   1:  PR[91,1] = PR[90,1] + -30.117;
   1:  PR[91,2] = PR[90,2] + 6.840;
   1:  PR[91,3] = PR[90,3] + 34.185;
   1:L PR[91] R[100]mm/sec CNT100;
   1:  PR[91,1] = PR[90,1] + -30.437;
   1:  PR[91,2] = PR[90,2] + 5.969;
   1:  PR[91,3] = PR[90,3] + 34.192;
   1:L PR[91] R[100]mm/sec CNT100;
   1:  PR[91,1] = PR[90,1] + -30.709;
   1:  PR[91,2] = PR[90,2] + 5.090;
   1:  PR[91,3] = PR[90,3] + 34.200;
   1:L PR[91] R[100]mm/sec CNT100;
   1:  PR[91,1] = PR[90,1] + -30.933;
   1:  PR[91,2] = PR[90,2] + 4.203;
   1:  PR[91,3] = PR[90,3] + 34.207;
   1:L PR[91] R[100]mm/sec CNT100;
   1:  PR[91,1] = PR[90,1] + -31.107;
   1:  PR[91,2] = PR[90,2] + 3.301;
   1:  PR[91,3] = PR[90,3] + 34.214;
   1:L PR[91] R[100]mm/sec CNT100;
   1:  PR[91,1] = PR[90,1] + -31.232;
   1:  PR[91,2] = PR[90,2] + 2.376;
   1:  PR[91,3] = PR[90,3] + 34.221;
   1:L PR[91] R[100]mm/sec CNT100;
   1:  PR[91,1] = PR[90,1] + -31.307;
   1:  PR[91,2] = PR[90,2] + 1.420;
   1:  PR[91,3] = PR[90,3] + 34.229;
   1:L PR[91] R[100]mm/sec CNT100;
   1:  PR[91,1] = PR[90,1] + -31.333;
   1:  PR[91,2] = PR[90,2] + 0.428;
   1:  PR[91,3] = PR[90,3] + 34.236;
   1:L PR[91] R[100]mm/sec CNT100;
   1:  PR[91,1] = PR[90,1] + -31.307;
   1:  PR[91,2] = PR[90,2] + -0.565;
   1:  PR[91,3] = PR[90,3] + 34.244;
   1:L PR[91] R[100]mm/sec CNT100;
   1:  PR[91,1] = PR[90,1] + -31.232;
   1:  PR[91,2] = PR[90,2] + -1.521;
   1:  PR[91,3] = PR[90,3] + 34.252;
   1:L PR[91] R[100]mm/sec CNT100;
   1:  PR[91,1] = PR[90,1] + -31.107;
   1:  PR[91,2] = PR[90,2] + -2.446;
   1:  PR[91,3] = PR[90,3] + 34.259;
   1:L PR[91] R[100]mm/sec CNT100;
   1:  PR[91,1] = PR[90,1] + -30.933;
   1:  PR[91,2] = PR[90,2] + -3.348;
   1:  PR[91,3] = PR[90,3] + 34.267;
   1:L PR[91] R[100]mm/sec CNT100;
   1:  PR[91,1] = PR[90,1] + -30.709;
   1:  PR[91,2] = PR[90,2] + -4.235;
   1:  PR[91,3] = PR[90,3] + 34.274;
   1:L PR[91] R[100]mm/sec CNT100;
   1:  PR[91,1] = PR[90,1] + -30.437;
   1:  PR[91,2] = PR[90,2] + -5.114;
   1:  PR[91,3] = PR[90,3] + 34.281;
   1:L PR[91] R[100]mm/sec CNT100;
   1:  PR[91,1] = PR[90,1] + -30.117;
   1:  PR[91,2] = PR[90,2] + -5.985;
   1:  PR[91,3] = PR[90,3] + 34.288;
   1:L PR[91] R[100]mm/sec CNT100;
   1:  PR[91,1] = PR[90,1] + -29.750;
   1:  PR[91,2] = PR[90,2] + -6.850;
   1:  PR[91,3] = PR[90,3] + 34.296;
   1:L PR[91] R[100]mm/sec CNT100;
   1:  PR[91,1] = PR[90,1] + -29.338;
   1:  PR[91,2] = PR[90,2] + -7.703;
   1:  PR[91,3] = PR[90,3] + 34.303;
   1:L PR[91] R[100]mm/sec CNT100;
   1:  PR[91,1] = PR[90,1] + -28.881;
   1:  PR[91,2] = PR[90,2] + -8.539;
   1:  PR[91,3] = PR[90,3] + 34.311;
   1:L PR[91] R[100]mm/sec CNT100;
   1:  PR[91,1] = PR[90,1] + -28.381;
   1:  PR[91,2] = PR[90,2] + -9.354;
   1:  PR[91,3] = PR[90,3] + 34.318;
   1:L PR[91] R[100]mm/sec CNT100;
   1:  PR[91,1] = PR[90,1] + -27.841;
   1:  PR[91,2] = PR[90,2] + -10.142;
   1:  PR[91,3] = PR[90,3] + 34.326;
   1:L PR[91] R[100]mm/sec CNT100;
   1:  PR[91,1] = PR[90,1] + -27.254;
   1:  PR[91,2] = PR[90,2] + -10.910;
   1:  PR[91,3] = PR[90,3] + 34.333;
   1:L PR[91] R[100]mm/sec CNT100;
   1:  PR[91,1] = PR[90,1] + -26.623;
   1:  PR[91,2] = PR[90,2] + -11.651;
   1:  PR[91,3] = PR[90,3] + 34.341;
   1:L PR[91] R[100]mm/sec CNT100;
   1:  PR[91,1] = PR[90,1] + -25.951;
   1:  PR[91,2] = PR[90,2] + -12.362;
   1:  PR[91,3] = PR[90,3] + 34.349;
   1:L PR[91] R[100]mm/sec CNT100;
   1:  PR[91,1] = PR[90,1] + -25.240;
   1:  PR[91,2] = PR[90,2] + -13.041;
   1:  PR[91,3] = PR[90,3] + 34.356;
   1:L PR[91] R[100]mm/sec CNT100;
   1:  PR[91,1] = PR[90,1] + -24.491;
   1:  PR[91,2] = PR[90,2] + -13.687;
   1:  PR[91,3] = PR[90,3] + 34.364;
   1:L PR[91] R[100]mm/sec CNT100;
   1:  PR[91,1] = PR[90,1] + -23.938;
   1:  PR[91,2] = PR[90,2] + -14.118;
   1:  PR[91,3] = PR[90,3] + 34.372;
   1:L PR[91] R[100]mm/sec CNT100;
   1:  PR[91,1] = PR[90,1] + -23.708;
   1:  PR[91,2] = PR[90,2] + -14.295;
   1:  PR[91,3] = PR[90,3] + 34.377;
   1:L PR[91] R[100]mm/sec CNT100;
   1:  PR[91,1] = PR[90,1] + -22.887;
   1:  PR[91,2] = PR[90,2] + -14.869;
   1:  PR[91,3] = PR[90,3] + 34.380;
   1:L PR[91] R[100]mm/sec CNT100;
   1:  PR[91,1] = PR[90,1] + -22.035;
   1:  PR[91,2] = PR[90,2] + -15.404;
   1:  PR[91,3] = PR[90,3] + 34.388;
   1:L PR[91] R[100]mm/sec CNT100;
   1:  PR[91,1] = PR[90,1] + -21.152;
   1:  PR[91,2] = PR[90,2] + -15.899;
   1:  PR[91,3] = PR[90,3] + 34.396;
   1:L PR[91] R[100]mm/sec CNT100;
   1:  PR[91,1] = PR[90,1] + -20.241;
   1:  PR[91,2] = PR[90,2] + -16.352;
   1:  PR[91,3] = PR[90,3] + 34.404;
   1:L PR[91] R[100]mm/sec CNT100;
   1:  PR[91,1] = PR[90,1] + -19.305;
   1:  PR[91,2] = PR[90,2] + -16.760;
   1:  PR[91,3] = PR[90,3] + 34.412;
   1:L PR[91] R[100]mm/sec CNT100;
   1:  PR[91,1] = PR[90,1] + -18.345;
   1:  PR[91,2] = PR[90,2] + -17.123;
   1:  PR[91,3] = PR[90,3] + 34.420;
   1:L PR[91] R[100]mm/sec CNT100;
   1:  PR[91,1] = PR[90,1] + -17.364;
   1:  PR[91,2] = PR[90,2] + -17.438;
   1:  PR[91,3] = PR[90,3] + 34.428;
   1:L PR[91] R[100]mm/sec CNT100;
   1:  PR[91,1] = PR[90,1] + -16.364;
   1:  PR[91,2] = PR[90,2] + -17.705;
   1:  PR[91,3] = PR[90,3] + 34.436;
   1:L PR[91] R[100]mm/sec CNT100;
   1:  PR[91,1] = PR[90,1] + -15.349;
   1:  PR[91,2] = PR[90,2] + -17.922;
   1:  PR[91,3] = PR[90,3] + 34.444;
   1:L PR[91] R[100]mm/sec CNT100;
   1:  PR[91,1] = PR[90,1] + -14.308;
   1:  PR[91,2] = PR[90,2] + -18.090;
   1:  PR[91,3] = PR[90,3] + 34.452;
   1:L PR[91] R[100]mm/sec CNT100;
   1:  PR[91,1] = PR[90,1] + -13.316;
   1:  PR[91,2] = PR[90,2] + -18.202;
   1:  PR[91,3] = PR[90,3] + 34.461;
   1:L PR[91] R[100]mm/sec CNT100;
   1:  PR[91,1] = PR[90,1] + -12.315;
   1:  PR[91,2] = PR[90,2] + -18.266;
   1:  PR[91,3] = PR[90,3] + 34.468;
   1:L PR[91] R[100]mm/sec CNT100;
   1:  PR[91,1] = PR[90,1] + -11.313;
   1:  PR[91,2] = PR[90,2] + -18.282;
   1:  PR[91,3] = PR[90,3] + 34.476;
   1:L PR[91] R[100]mm/sec CNT100;
   1:  PR[91,1] = PR[90,1] + -10.312;
   1:  PR[91,2] = PR[90,2] + -18.250;
   1:  PR[91,3] = PR[90,3] + 34.484;
   1:L PR[91] R[100]mm/sec CNT100;
   1:  PR[91,1] = PR[90,1] + -9.313;
   1:  PR[91,2] = PR[90,2] + -18.169;
   1:  PR[91,3] = PR[90,3] + 34.492;
   1:L PR[91] R[100]mm/sec CNT100;
   1:  PR[91,1] = PR[90,1] + -8.321;
   1:  PR[91,2] = PR[90,2] + -18.039;
   1:  PR[91,3] = PR[90,3] + 34.500;
   1:L PR[91] R[100]mm/sec CNT100;
   1:  PR[91,1] = PR[90,1] + -7.337;
   1:  PR[91,2] = PR[90,2] + -17.862;
   1:  PR[91,3] = PR[90,3] + 34.508;
   1:L PR[91] R[100]mm/sec CNT100;
   1:  PR[91,1] = PR[90,1] + -6.364;
   1:  PR[91,2] = PR[90,2] + -17.636;
   1:  PR[91,3] = PR[90,3] + 34.516;
   1:L PR[91] R[100]mm/sec CNT100;
   1:  PR[91,1] = PR[90,1] + -5.403;
   1:  PR[91,2] = PR[90,2] + -17.363;
   1:  PR[91,3] = PR[90,3] + 34.524;
   1:L PR[91] R[100]mm/sec CNT100;
   1:  PR[91,1] = PR[90,1] + -4.840;
   1:  PR[91,2] = PR[90,2] + -17.177;
   1:  PR[91,3] = PR[90,3] + 34.532;
   1:L PR[91] R[100]mm/sec CNT100;
   1:  PR[91,1] = PR[90,1] + -3.848;
   1:  PR[91,2] = PR[90,2] + -16.806;
   1:  PR[91,3] = PR[90,3] + 34.536;
   1:L PR[91] R[100]mm/sec CNT100;
   1:  PR[91,1] = PR[90,1] + -2.883;
   1:  PR[91,2] = PR[90,2] + -16.387;
   1:  PR[91,3] = PR[90,3] + 34.545;
   1:L PR[91] R[100]mm/sec CNT100;
   1:  PR[91,1] = PR[90,1] + -1.942;
   1:  PR[91,2] = PR[90,2] + -15.918;
   1:  PR[91,3] = PR[90,3] + 34.553;
   1:L PR[91] R[100]mm/sec CNT100;
   1:  PR[91,1] = PR[90,1] + -1.554;
   1:  PR[91,2] = PR[90,2] + -15.705;
   1:  PR[91,3] = PR[90,3] + 34.561;
   1:L PR[91] R[100]mm/sec CNT100;
   1:  PR[91,1] = PR[90,1] + -1.132;
   1:  PR[91,2] = PR[90,2] + -15.511;
   1:  PR[91,3] = PR[90,3] + 34.565;
   1:L PR[91] R[100]mm/sec CNT100;
   1:  PR[91,1] = PR[90,1] + -0.658;
   1:  PR[91,2] = PR[90,2] + -15.382;
   1:  PR[91,3] = PR[90,3] + 34.568;
   1:L PR[91] R[100]mm/sec CNT100;
   1:  PR[91,1] = PR[90,1] + -0.170;
   1:  PR[91,2] = PR[90,2] + -15.334;
   1:  PR[91,3] = PR[90,3] + 34.572;
   1:L PR[91] R[100]mm/sec CNT100;
   1:  PR[91,1] = PR[90,1] + 0.322;
   1:  PR[91,2] = PR[90,2] + -15.366;
   1:  PR[91,3] = PR[90,3] + 34.576;
   1:L PR[91] R[100]mm/sec CNT100;
   1:  PR[91] = PR[90];
   1:  PR[91,1] = PR[90,1] + 0.880;
   1:  PR[91,2] = PR[90,2] + -15.981;
   1:  PR[91,3] = PR[90,3] + 35.910;
   1:L PR[91] R[100]mm/sec CNT100;
   1:  PR[91,1] = PR[90,1] + 1.236;
   1:  PR[91,2] = PR[90,2] + -16.136;
   1:  PR[91,3] = PR[90,3] + 34.584;
   1:L PR[91] R[100]mm/sec CNT100;
   1:  PR[91,1] = PR[90,1] + 1.910;
   1:  PR[91,2] = PR[90,2] + -16.474;
   1:  PR[91,3] = PR[90,3] + 34.587;
   1:L PR[91] R[100]mm/sec CNT100;
   1:  PR[91,1] = PR[90,1] + 2.739;
   1:  PR[91,2] = PR[90,2] + -16.844;
   1:  PR[91,3] = PR[90,3] + 34.593;
   1:L PR[91] R[100]mm/sec CNT100;
   1:  PR[91,1] = PR[90,1] + 3.804;
   1:  PR[91,2] = PR[90,2] + -17.258;
   1:  PR[91,3] = PR[90,3] + 34.600;
   1:L PR[91] R[100]mm/sec CNT100;
   1:  PR[91,1] = PR[90,1] + 4.756;
   1:  PR[91,2] = PR[90,2] + -17.571;
   1:  PR[91,3] = PR[90,3] + 34.609;
   1:L PR[91] R[100]mm/sec CNT100;
   1:  PR[91,1] = PR[90,1] + 5.722;
   1:  PR[91,2] = PR[90,2] + -17.837;
   1:  PR[91,3] = PR[90,3] + 34.617;
   1:L PR[91] R[100]mm/sec CNT100;
   1:  PR[91,1] = PR[90,1] + 6.804;
   1:  PR[91,2] = PR[90,2] + -18.077;
   1:  PR[91,3] = PR[90,3] + 34.625;
   1:L PR[91] R[100]mm/sec CNT100;
   1:  PR[91,1] = PR[90,1] + 7.689;
   1:  PR[91,2] = PR[90,2] + -18.229;
   1:  PR[91,3] = PR[90,3] + 34.634;
   1:L PR[91] R[100]mm/sec CNT100;
   1:  PR[91,1] = PR[90,1] + 8.683;
   1:  PR[91,2] = PR[90,2] + -18.352;
   1:  PR[91,3] = PR[90,3] + 34.641;
   1:L PR[91] R[100]mm/sec CNT100;
   1:  PR[91,1] = PR[90,1] + 9.992;
   1:  PR[91,2] = PR[90,2] + -18.438;
   1:  PR[91,3] = PR[90,3] + 34.649;
   1:L PR[91] R[100]mm/sec CNT100;
   1:  PR[91,1] = PR[90,1] + 10.692;
   1:  PR[91,2] = PR[90,2] + -18.454;
   1:  PR[91,3] = PR[90,3] + 34.660;
   1:L PR[91] R[100]mm/sec CNT100;
   1:  PR[91,1] = PR[90,1] + 11.698;
   1:  PR[91,2] = PR[90,2] + -18.431;
   1:  PR[91,3] = PR[90,3] + 34.665;
   1:L PR[91] R[100]mm/sec CNT100;
   1:  PR[91,1] = PR[90,1] + 12.702;
   1:  PR[91,2] = PR[90,2] + -18.360;
   1:  PR[91,3] = PR[90,3] + 34.673;
   1:L PR[91] R[100]mm/sec CNT100;
   1:  PR[91,1] = PR[90,1] + 13.700;
   1:  PR[91,2] = PR[90,2] + -18.241;
   1:  PR[91,3] = PR[90,3] + 34.681;
   1:L PR[91] R[100]mm/sec CNT100;
   1:  PR[91,1] = PR[90,1] + 14.691;
   1:  PR[91,2] = PR[90,2] + -18.073;
   1:  PR[91,3] = PR[90,3] + 34.689;
   1:L PR[91] R[100]mm/sec CNT100;
   1:  PR[91,1] = PR[90,1] + 15.673;
   1:  PR[91,2] = PR[90,2] + -17.858;
   1:  PR[91,3] = PR[90,3] + 34.697;
   1:L PR[91] R[100]mm/sec CNT100;
   1:  PR[91,1] = PR[90,1] + 16.643;
   1:  PR[91,2] = PR[90,2] + -17.595;
   1:  PR[91,3] = PR[90,3] + 34.705;
   1:L PR[91] R[100]mm/sec CNT100;
   1:  PR[91,1] = PR[90,1] + 17.597;
   1:  PR[91,2] = PR[90,2] + -17.287;
   1:  PR[91,3] = PR[90,3] + 34.713;
   1:L PR[91] R[100]mm/sec CNT100;
   1:  PR[91,1] = PR[90,1] + 18.535;
   1:  PR[91,2] = PR[90,2] + -16.932;
   1:  PR[91,3] = PR[90,3] + 34.721;
   1:L PR[91] R[100]mm/sec CNT100;
   1:  PR[91,1] = PR[90,1] + 19.454;
   1:  PR[91,2] = PR[90,2] + -16.534;
   1:  PR[91,3] = PR[90,3] + 34.729;
   1:L PR[91] R[100]mm/sec CNT100;
   1:  PR[91,1] = PR[90,1] + 20.350;
   1:  PR[91,2] = PR[90,2] + -16.093;
   1:  PR[91,3] = PR[90,3] + 34.737;
   1:L PR[91] R[100]mm/sec CNT100;
   1:  PR[91,1] = PR[90,1] + 21.242;
   1:  PR[91,2] = PR[90,2] + -15.600;
   1:  PR[91,3] = PR[90,3] + 34.745;
   1:L PR[91] R[100]mm/sec CNT100;
   1:  PR[91,1] = PR[90,1] + 22.108;
   1:  PR[91,2] = PR[90,2] + -15.063;
   1:  PR[91,3] = PR[90,3] + 34.753;
   1:L PR[91] R[100]mm/sec CNT100;
   1:  PR[91,1] = PR[90,1] + 22.940;
   1:  PR[91,2] = PR[90,2] + -14.487;
   1:  PR[91,3] = PR[90,3] + 34.761;
   1:L PR[91] R[100]mm/sec CNT100;
   1:  PR[91,1] = PR[90,1] + 23.738;
   1:  PR[91,2] = PR[90,2] + -13.872;
   1:  PR[91,3] = PR[90,3] + 34.769;
   1:L PR[91] R[100]mm/sec CNT100;
   1:  PR[91,1] = PR[90,1] + 24.292;
   1:  PR[91,2] = PR[90,2] + -13.400;
   1:  PR[91,3] = PR[90,3] + 34.777;
   1:L PR[91] R[100]mm/sec CNT100;
   1:  PR[91,1] = PR[90,1] + 25.224;
   1:  PR[91,2] = PR[90,2] + -12.533;
   1:  PR[91,3] = PR[90,3] + 34.783;
   1:L PR[91] R[100]mm/sec CNT100;
   1:  PR[91,1] = PR[90,1] + 25.905;
   1:  PR[91,2] = PR[90,2] + -11.814;
   1:  PR[91,3] = PR[90,3] + 34.793;
   1:L PR[91] R[100]mm/sec CNT100;
   1:  PR[91,1] = PR[90,1] + 26.547;
   1:  PR[91,2] = PR[90,2] + -11.061;
   1:  PR[91,3] = PR[90,3] + 34.801;
   1:L PR[91] R[100]mm/sec CNT100;
   1:  PR[91,1] = PR[90,1] + 27.147;
   1:  PR[91,2] = PR[90,2] + -10.279;
   1:  PR[91,3] = PR[90,3] + 34.809;
   1:L PR[91] R[100]mm/sec CNT100;
   1:  PR[91,1] = PR[90,1] + 27.703;
   1:  PR[91,2] = PR[90,2] + -9.470;
   1:  PR[91,3] = PR[90,3] + 34.817;
   1:L PR[91] R[100]mm/sec CNT100;
   1:  PR[91,1] = PR[90,1] + 28.215;
   1:  PR[91,2] = PR[90,2] + -8.638;
   1:  PR[91,3] = PR[90,3] + 34.825;
   1:L PR[91] R[100]mm/sec CNT100;
   1:  PR[91,1] = PR[90,1] + 28.681;
   1:  PR[91,2] = PR[90,2] + -7.788;
   1:  PR[91,3] = PR[90,3] + 34.833;
   1:L PR[91] R[100]mm/sec CNT100;
   1:  PR[91,1] = PR[90,1] + 29.101;
   1:  PR[91,2] = PR[90,2] + -6.925;
   1:  PR[91,3] = PR[90,3] + 34.840;
   1:L PR[91] R[100]mm/sec CNT100;
   1:  PR[91,1] = PR[90,1] + 29.472;
   1:  PR[91,2] = PR[90,2] + -6.053;
   1:  PR[91,3] = PR[90,3] + 34.848;
   1:L PR[91] R[100]mm/sec CNT100;
   1:  PR[91,1] = PR[90,1] + 29.795;
   1:  PR[91,2] = PR[90,2] + -5.175;
   1:  PR[91,3] = PR[90,3] + 34.855;
   1:L PR[91] R[100]mm/sec CNT100;
   1:  PR[91,1] = PR[90,1] + 30.069;
   1:  PR[91,2] = PR[90,2] + -4.288;
   1:  PR[91,3] = PR[90,3] + 34.863;
   1:L PR[91] R[100]mm/sec CNT100;
   1:  PR[91,1] = PR[90,1] + 30.293;
   1:  PR[91,2] = PR[90,2] + -3.390;
   1:  PR[91,3] = PR[90,3] + 34.870;
   1:L PR[91] R[100]mm/sec CNT100;
   1:  PR[91,1] = PR[90,1] + 30.468;
   1:  PR[91,2] = PR[90,2] + -2.475;
   1:  PR[91,3] = PR[90,3] + 34.878;
   1:L PR[91] R[100]mm/sec CNT100;
   1:  PR[91,1] = PR[90,1] + 30.593;
   1:  PR[91,2] = PR[90,2] + -1.537;
   1:  PR[91,3] = PR[90,3] + 34.885;
   1:L PR[91] R[100]mm/sec CNT100;
   1:  PR[91,1] = PR[90,1] + 30.669;
   1:  PR[91,2] = PR[90,2] + -0.572;
   1:  PR[91,3] = PR[90,3] + 34.893;
   1:L PR[91] R[100]mm/sec CNT100;
   1:  PR[91,1] = PR[90,1] + 30.692;
   1:  PR[91,2] = PR[90,2] + 0.428;
   1:  PR[91,3] = PR[90,3] + 34.900;
   1:L PR[91] R[100]mm/sec CNT100;
   1:  PR[91,1] = PR[90,1] + 30.669;
   1:  PR[91,2] = PR[90,2] + 1.427;
   1:  PR[91,3] = PR[90,3] + 34.908;
   1:L PR[91] R[100]mm/sec CNT100;
   1:  PR[91,1] = PR[90,1] + 30.593;
   1:  PR[91,2] = PR[90,2] + 2.392;
   1:  PR[91,3] = PR[90,3] + 34.916;
   1:L PR[91] R[100]mm/sec CNT100;
   1:  PR[91,1] = PR[90,1] + 30.468;
   1:  PR[91,2] = PR[90,2] + 3.330;
   1:  PR[91,3] = PR[90,3] + 34.924;
   1:L PR[91] R[100]mm/sec CNT100;
   1:  PR[91,1] = PR[90,1] + 30.293;
   1:  PR[91,2] = PR[90,2] + 4.245;
   1:  PR[91,3] = PR[90,3] + 34.931;
   1:L PR[91] R[100]mm/sec CNT100;
   1:  PR[91,1] = PR[90,1] + 30.069;
   1:  PR[91,2] = PR[90,2] + 5.143;
   1:  PR[91,3] = PR[90,3] + 34.939;
   1:L PR[91] R[100]mm/sec CNT100;
   1:  PR[91,1] = PR[90,1] + 29.795;
   1:  PR[91,2] = PR[90,2] + 6.030;
   1:  PR[91,3] = PR[90,3] + 34.946;
   1:L PR[91] R[100]mm/sec CNT100;
   1:  PR[91,1] = PR[90,1] + 29.472;
   1:  PR[91,2] = PR[90,2] + 6.909;
   1:  PR[91,3] = PR[90,3] + 34.954;
   1:L PR[91] R[100]mm/sec CNT100;
   1:  PR[91,1] = PR[90,1] + 29.101;
   1:  PR[91,2] = PR[90,2] + 7.780;
   1:  PR[91,3] = PR[90,3] + 34.961;
   1:L PR[91] R[100]mm/sec CNT100;
   1:  PR[91,1] = PR[90,1] + 28.681;
   1:  PR[91,2] = PR[90,2] + 8.644;
   1:  PR[91,3] = PR[90,3] + 34.969;
   1:L PR[91] R[100]mm/sec CNT100;
   1:  PR[91,1] = PR[90,1] + 28.215;
   1:  PR[91,2] = PR[90,2] + 9.493;
   1:  PR[91,3] = PR[90,3] + 34.976;
   1:L PR[91] R[100]mm/sec CNT100;
   1:  PR[91,1] = PR[90,1] + 27.703;
   1:  PR[91,2] = PR[90,2] + 10.326;
   1:  PR[91,3] = PR[90,3] + 34.984;
   1:L PR[91] R[100]mm/sec CNT100;
   1:  PR[91,1] = PR[90,1] + 27.423;
   1:  PR[91,2] = PR[90,2] + 10.735;
   1:  PR[91,3] = PR[90,3] + 34.992;
   1:L PR[91] R[100]mm/sec CNT100;
   1:  PR[91,1] = PR[90,1] + 27.148;
   1:  PR[91,2] = PR[90,2] + 11.133;
   1:  PR[91,3] = PR[90,3] + 34.996;
   1:L PR[91] R[100]mm/sec CNT100;
   1:  PR[91,1] = PR[90,1] + 26.547;
   1:  PR[91,2] = PR[90,2] + 11.916;
   1:  PR[91,3] = PR[90,3] + 35.000;
   1:L PR[91] R[100]mm/sec CNT100;
   1:  PR[91,1] = PR[90,1] + 25.905;
   1:  PR[91,2] = PR[90,2] + 12.669;
   1:  PR[91,3] = PR[90,3] + 35.007;
   1:L PR[91] R[100]mm/sec CNT100;
   1:  PR[91,1] = PR[90,1] + 25.224;
   1:  PR[91,2] = PR[90,2] + 13.388;
   1:  PR[91,3] = PR[90,3] + 35.015;
   1:L PR[91] R[100]mm/sec CNT100;
   1:  PR[91,1] = PR[90,1] + 24.292;
   1:  PR[91,2] = PR[90,2] + 14.256;
   1:  PR[91,3] = PR[90,3] + 35.023;
   1:L PR[91] R[100]mm/sec CNT100;
   1:  PR[91,1] = PR[90,1] + 23.738;
   1:  PR[91,2] = PR[90,2] + 14.727;
   1:  PR[91,3] = PR[90,3] + 35.033;
   1:L PR[91] R[100]mm/sec CNT100;
   1:  PR[91,1] = PR[90,1] + 22.940;
   1:  PR[91,2] = PR[90,2] + 15.342;
   1:  PR[91,3] = PR[90,3] + 35.039;
   1:L PR[91] R[100]mm/sec CNT100;
   1:  PR[91,1] = PR[90,1] + 22.108;
   1:  PR[91,2] = PR[90,2] + 15.918;
   1:  PR[91,3] = PR[90,3] + 35.047;
   1:L PR[91] R[100]mm/sec CNT100;
   1:  PR[91,1] = PR[90,1] + 21.242;
   1:  PR[91,2] = PR[90,2] + 16.455;
   1:  PR[91,3] = PR[90,3] + 35.055;
   1:L PR[91] R[100]mm/sec CNT100;
   1:  PR[91,1] = PR[90,1] + 20.339;
   1:  PR[91,2] = PR[90,2] + 16.954;
   1:  PR[91,3] = PR[90,3] + 35.063;
   1:L PR[91] R[100]mm/sec CNT100;
   1:  PR[91,1] = PR[90,1] + 19.454;
   1:  PR[91,2] = PR[90,2] + 17.389;
   1:  PR[91,3] = PR[90,3] + 35.072;
   1:L PR[91] R[100]mm/sec CNT100;
   1:  PR[91,1] = PR[90,1] + 18.535;
   1:  PR[91,2] = PR[90,2] + 17.788;
   1:  PR[91,3] = PR[90,3] + 35.079;
   1:L PR[91] R[100]mm/sec CNT100;
   1:  PR[91,1] = PR[90,1] + 17.597;
   1:  PR[91,2] = PR[90,2] + 18.142;
   1:  PR[91,3] = PR[90,3] + 35.087;
   1:L PR[91] R[100]mm/sec CNT100;
   1:  PR[91,1] = PR[90,1] + 16.642;
   1:  PR[91,2] = PR[90,2] + 18.451;
   1:  PR[91,3] = PR[90,3] + 35.095;
   1:L PR[91] R[100]mm/sec CNT100;
   1:  PR[91,1] = PR[90,1] + 15.673;
   1:  PR[91,2] = PR[90,2] + 18.713;
   1:  PR[91,3] = PR[90,3] + 35.103;
   1:L PR[91] R[100]mm/sec CNT100;
   1:  PR[91,1] = PR[90,1] + 14.691;
   1:  PR[91,2] = PR[90,2] + 18.929;
   1:  PR[91,3] = PR[90,3] + 35.111;
   1:L PR[91] R[100]mm/sec CNT100;
   1:  PR[91,1] = PR[90,1] + 13.698;
   1:  PR[91,2] = PR[90,2] + 19.096;
   1:  PR[91,3] = PR[90,3] + 35.119;
   1:L PR[91] R[100]mm/sec CNT100;
   1:  PR[91,1] = PR[90,1] + 13.203;
   1:  PR[91,2] = PR[90,2] + 19.159;
   1:  PR[91,3] = PR[90,3] + 35.127;
   1:L PR[91] R[100]mm/sec CNT100;
   1:  PR[91,1] = PR[90,1] + 12.701;
   1:  PR[91,2] = PR[90,2] + 19.215;
   1:  PR[91,3] = PR[90,3] + 35.131;
   1:L PR[91] R[100]mm/sec CNT100;
   1:  PR[91,1] = PR[90,1] + 12.138;
   1:  PR[91,2] = PR[90,2] + 19.258;
   1:  PR[91,3] = PR[90,3] + 35.135;
   1:L PR[91] R[100]mm/sec CNT100;
   1:  PR[91,1] = PR[90,1] + 11.052;
   1:  PR[91,2] = PR[90,2] + 19.304;
   1:  PR[91,3] = PR[90,3] + 35.140;
   1:L PR[91] R[100]mm/sec CNT100;
   1:  PR[91,1] = PR[90,1] + 10.694;
   1:  PR[91,2] = PR[90,2] + 19.309;
   1:  PR[91,3] = PR[90,3] + 35.148;
   1:L PR[91] R[100]mm/sec CNT100;
   1:  PR[91,1] = PR[90,1] + 9.685;
   1:  PR[91,2] = PR[90,2] + 19.283;
   1:  PR[91,3] = PR[90,3] + 35.151;
   1:L PR[91] R[100]mm/sec CNT100;
   1:  PR[91,1] = PR[90,1] + 8.920;
   1:  PR[91,2] = PR[90,2] + 19.228;
   1:  PR[91,3] = PR[90,3] + 35.159;
   1:L PR[91] R[100]mm/sec CNT100;
   1:  PR[91,1] = PR[90,1] + 7.686;
   1:  PR[91,2] = PR[90,2] + 19.084;
   1:  PR[91,3] = PR[90,3] + 35.165;
   1:L PR[91] R[100]mm/sec CNT100;
   1:  PR[91,1] = PR[90,1] + 6.699;
   1:  PR[91,2] = PR[90,2] + 18.912;
   1:  PR[91,3] = PR[90,3] + 35.175;
   1:L PR[91] R[100]mm/sec CNT100;
   1:  PR[91,1] = PR[90,1] + 5.721;
   1:  PR[91,2] = PR[90,2] + 18.692;
   1:  PR[91,3] = PR[90,3] + 35.183;
   1:L PR[91] R[100]mm/sec CNT100;
   1:  PR[91,1] = PR[90,1] + 4.734;
   1:  PR[91,2] = PR[90,2] + 18.419;
   1:  PR[91,3] = PR[90,3] + 35.191;
   1:L PR[91] R[100]mm/sec CNT100;
   1:  PR[91,1] = PR[90,1] + 3.800;
   1:  PR[91,2] = PR[90,2] + 18.112;
   1:  PR[91,3] = PR[90,3] + 35.199;
   1:L PR[91] R[100]mm/sec CNT100;
   1:  PR[91,1] = PR[90,1] + 2.864;
   1:  PR[91,2] = PR[90,2] + 17.752;
   1:  PR[91,3] = PR[90,3] + 35.207;
   1:L PR[91] R[100]mm/sec CNT100;
   1:  PR[91,1] = PR[90,1] + 1.949;
   1:  PR[91,2] = PR[90,2] + 17.348;
   1:  PR[91,3] = PR[90,3] + 35.215;
   1:L PR[91] R[100]mm/sec CNT100;
   1:  PR[91,1] = PR[90,1] + 1.236;
   1:  PR[91,2] = PR[90,2] + 16.992;
   1:  PR[91,3] = PR[90,3] + 35.223;
   1:L PR[91] R[100]mm/sec CNT100;
   1:  PR[91,1] = PR[90,1] + 0.880;
   1:  PR[91,2] = PR[90,2] + 16.836;
   1:  PR[91,3] = PR[90,3] + 35.230;
   1:L PR[91] R[100]mm/sec CNT100;
   1:  PR[91,1] = PR[90,1] + 0.406;
   1:  PR[91,2] = PR[90,2] + 16.707;
   1:  PR[91,3] = PR[90,3] + 35.233;
   1:L PR[91] R[100]mm/sec CNT100;
   1:  PR[91,1] = PR[90,1] + -0.086;
   1:  PR[91,2] = PR[90,2] + 16.662;
   1:  PR[91,3] = PR[90,3] + 35.237;
   1:L PR[91] R[100]mm/sec CNT100;
   1:  PR[91,1] = PR[90,1] + -0.574;
   1:  PR[91,2] = PR[90,2] + 16.697;
   1:  PR[91,3] = PR[90,3] + 35.241;
   1:L PR[91] R[100]mm/sec CNT100;
   1:  PR[91,1] = PR[90,1] + -1.051;
   1:  PR[91,2] = PR[90,2] + 16.812;
   1:  PR[91,3] = PR[90,3] + 35.244;
   1:L PR[91] R[100]mm/sec CNT100;
   1:  PR[91,1] = PR[90,1] + -1.476;
   1:  PR[91,2] = PR[90,2] + 16.991;
   1:  PR[91,3] = PR[90,3] + 35.248;
   1:L PR[91] R[100]mm/sec CNT100;
   1:  PR[91,1] = PR[90,1] + -2.136;
   1:  PR[91,2] = PR[90,2] + 17.322;
   1:  PR[91,3] = PR[90,3] + 35.252;
   1:L PR[91] R[100]mm/sec CNT100;
   1:  PR[91,1] = PR[90,1] + -2.980;
   1:  PR[91,2] = PR[90,2] + 17.700;
   1:  PR[91,3] = PR[90,3] + 35.258;
   1:L PR[91] R[100]mm/sec CNT100;
   1:  PR[91,1] = PR[90,1] + -4.044;
   1:  PR[91,2] = PR[90,2] + 18.115;
   1:  PR[91,3] = PR[90,3] + 35.265;
   1:L PR[91] R[100]mm/sec CNT100;
   1:  PR[91,1] = PR[90,1] + -4.996;
   1:  PR[91,2] = PR[90,2] + 18.428;
   1:  PR[91,3] = PR[90,3] + 35.274;
   1:L PR[91] R[100]mm/sec CNT100;
   1:  PR[91,1] = PR[90,1] + -5.962;
   1:  PR[91,2] = PR[90,2] + 18.694;
   1:  PR[91,3] = PR[90,3] + 35.282;
   1:L PR[91] R[100]mm/sec CNT100;
   1:  PR[91,1] = PR[90,1] + -7.044;
   1:  PR[91,2] = PR[90,2] + 18.933;
   1:  PR[91,3] = PR[90,3] + 35.290;
   1:L PR[91] R[100]mm/sec CNT100;
   1:  PR[91,1] = PR[90,1] + -7.929;
   1:  PR[91,2] = PR[90,2] + 19.085;
   1:  PR[91,3] = PR[90,3] + 35.299;
   1:L PR[91] R[100]mm/sec CNT100;
   1:  PR[91,1] = PR[90,1] + -8.924;
   1:  PR[91,2] = PR[90,2] + 19.208;
   1:  PR[91,3] = PR[90,3] + 35.306;
   1:L PR[91] R[100]mm/sec CNT100;
   1:  PR[91,1] = PR[90,1] + -10.233;
   1:  PR[91,2] = PR[90,2] + 19.293;
   1:  PR[91,3] = PR[90,3] + 35.314;
   1:L PR[91] R[100]mm/sec CNT100;
   1:  PR[91,1] = PR[90,1] + -10.933;
   1:  PR[91,2] = PR[90,2] + 19.309;
   1:  PR[91,3] = PR[90,3] + 35.325;
   1:L PR[91] R[100]mm/sec CNT100;
   1:  PR[91,1] = PR[90,1] + -11.939;
   1:  PR[91,2] = PR[90,2] + 19.286;
   1:  PR[91,3] = PR[90,3] + 35.330;
   1:L PR[91] R[100]mm/sec CNT100;
   1:  PR[91,1] = PR[90,1] + -12.943;
   1:  PR[91,2] = PR[90,2] + 19.215;
   1:  PR[91,3] = PR[90,3] + 35.338;
   1:L PR[91] R[100]mm/sec CNT100;
   1:  PR[91,1] = PR[90,1] + -13.941;
   1:  PR[91,2] = PR[90,2] + 19.095;
   1:  PR[91,3] = PR[90,3] + 35.346;
   1:L PR[91] R[100]mm/sec CNT100;
   1:  PR[91,1] = PR[90,1] + -14.933;
   1:  PR[91,2] = PR[90,2] + 18.928;
   1:  PR[91,3] = PR[90,3] + 35.354;
   1:L PR[91] R[100]mm/sec CNT100;
   1:  PR[91,1] = PR[90,1] + -15.916;
   1:  PR[91,2] = PR[90,2] + 18.713;
   1:  PR[91,3] = PR[90,3] + 35.362;
   1:L PR[91] R[100]mm/sec CNT100;
   1:  PR[91,1] = PR[90,1] + -16.602;
   1:  PR[91,2] = PR[90,2] + 18.530;
   1:  PR[91,3] = PR[90,3] + 35.370;
   1:L PR[91] R[100]mm/sec CNT100;
   1:  PR[91,1] = PR[90,1] + -17.842;
   1:  PR[91,2] = PR[90,2] + 18.141;
   1:  PR[91,3] = PR[90,3] + 35.376;
   1:L PR[91] R[100]mm/sec CNT100;
   1:  PR[91,1] = PR[90,1] + -18.635;
   1:  PR[91,2] = PR[90,2] + 17.843;
   1:  PR[91,3] = PR[90,3] + 35.386;
   1:L PR[91] R[100]mm/sec CNT100;
   1:  PR[91,1] = PR[90,1] + -19.695;
   1:  PR[91,2] = PR[90,2] + 17.388;
   1:  PR[91,3] = PR[90,3] + 35.393;
   1:L PR[91] R[100]mm/sec CNT100;
   1:  PR[91,1] = PR[90,1] + -20.591;
   1:  PR[91,2] = PR[90,2] + 16.946;
   1:  PR[91,3] = PR[90,3] + 35.402;
   1:L PR[91] R[100]mm/sec CNT100;
   1:  PR[91,1] = PR[90,1] + -21.482;
   1:  PR[91,2] = PR[90,2] + 16.452;
   1:  PR[91,3] = PR[90,3] + 35.410;
   1:L PR[91] R[100]mm/sec CNT100;
   1:  PR[91,1] = PR[90,1] + -22.348;
   1:  PR[91,2] = PR[90,2] + 15.914;
   1:  PR[91,3] = PR[90,3] + 35.418;
   1:L PR[91] R[100]mm/sec CNT100;
   1:  PR[91,1] = PR[90,1] + -23.180;
   1:  PR[91,2] = PR[90,2] + 15.338;
   1:  PR[91,3] = PR[90,3] + 35.426;
   1:L PR[91] R[100]mm/sec CNT100;
   1:  PR[91,1] = PR[90,1] + -23.978;
   1:  PR[91,2] = PR[90,2] + 14.723;
   1:  PR[91,3] = PR[90,3] + 35.434;
   1:L PR[91] R[100]mm/sec CNT100;
   1:  PR[91,1] = PR[90,1] + -24.739;
   1:  PR[91,2] = PR[90,2] + 14.073;
   1:  PR[91,3] = PR[90,3] + 35.442;
   1:L PR[91] R[100]mm/sec CNT100;
   1:  PR[91,1] = PR[90,1] + -25.462;
   1:  PR[91,2] = PR[90,2] + 13.388;
   1:  PR[91,3] = PR[90,3] + 35.450;
   1:L PR[91] R[100]mm/sec CNT100;
   1:  PR[91,1] = PR[90,1] + -26.146;
   1:  PR[91,2] = PR[90,2] + 12.670;
   1:  PR[91,3] = PR[90,3] + 35.458;
   1:L PR[91] R[100]mm/sec CNT100;
   1:  PR[91,1] = PR[90,1] + -26.787;
   1:  PR[91,2] = PR[90,2] + 11.921;
   1:  PR[91,3] = PR[90,3] + 35.466;
   1:L PR[91] R[100]mm/sec CNT100;
   1:  PR[91,1] = PR[90,1] + -27.387;
   1:  PR[91,2] = PR[90,2] + 11.141;
   1:  PR[91,3] = PR[90,3] + 35.474;
   1:L PR[91] R[100]mm/sec CNT100;
   1:  PR[91,1] = PR[90,1] + -27.942;
   1:  PR[91,2] = PR[90,2] + 10.333;
   1:  PR[91,3] = PR[90,3] + 35.482;
   1:L PR[91] R[100]mm/sec CNT100;
   1:  PR[91,1] = PR[90,1] + -28.453;
   1:  PR[91,2] = PR[90,2] + 9.500;
   1:  PR[91,3] = PR[90,3] + 35.490;
   1:L PR[91] R[100]mm/sec CNT100;
   1:  PR[91,1] = PR[90,1] + -28.919;
   1:  PR[91,2] = PR[90,2] + 8.647;
   1:  PR[91,3] = PR[90,3] + 35.498;
   1:L PR[91] R[100]mm/sec CNT100;
   1:  PR[91,1] = PR[90,1] + -29.339;
   1:  PR[91,2] = PR[90,2] + 7.778;
   1:  PR[91,3] = PR[90,3] + 35.505;
   1:L PR[91] R[100]mm/sec CNT100;
   1:  PR[91,1] = PR[90,1] + -29.710;
   1:  PR[91,2] = PR[90,2] + 6.900;
   1:  PR[91,3] = PR[90,3] + 35.513;
   1:L PR[91] R[100]mm/sec CNT100;
   1:  PR[91,1] = PR[90,1] + -30.033;
   1:  PR[91,2] = PR[90,2] + 6.016;
   1:  PR[91,3] = PR[90,3] + 35.521;
   1:L PR[91] R[100]mm/sec CNT100;
   1:  PR[91,1] = PR[90,1] + -30.307;
   1:  PR[91,2] = PR[90,2] + 5.126;
   1:  PR[91,3] = PR[90,3] + 35.528;
   1:L PR[91] R[100]mm/sec CNT100;
   1:  PR[91,1] = PR[90,1] + -30.532;
   1:  PR[91,2] = PR[90,2] + 4.229;
   1:  PR[91,3] = PR[90,3] + 35.535;
   1:L PR[91] R[100]mm/sec CNT100;
   1:  PR[91,1] = PR[90,1] + -30.707;
   1:  PR[91,2] = PR[90,2] + 3.318;
   1:  PR[91,3] = PR[90,3] + 35.543;
   1:L PR[91] R[100]mm/sec CNT100;
   1:  PR[91,1] = PR[90,1] + -30.832;
   1:  PR[91,2] = PR[90,2] + 2.386;
   1:  PR[91,3] = PR[90,3] + 35.550;
   1:L PR[91] R[100]mm/sec CNT100;
   1:  PR[91,1] = PR[90,1] + -30.907;
   1:  PR[91,2] = PR[90,2] + 1.425;
   1:  PR[91,3] = PR[90,3] + 35.558;
   1:L PR[91] R[100]mm/sec CNT100;
   1:  PR[91,1] = PR[90,1] + -30.931;
   1:  PR[91,2] = PR[90,2] + 0.428;
   1:  PR[91,3] = PR[90,3] + 35.565;
   1:L PR[91] R[100]mm/sec CNT100;
   1:  PR[91,1] = PR[90,1] + -30.907;
   1:  PR[91,2] = PR[90,2] + -0.570;
   1:  PR[91,3] = PR[90,3] + 35.573;
   1:L PR[91] R[100]mm/sec CNT100;
   1:  PR[91,1] = PR[90,1] + -30.832;
   1:  PR[91,2] = PR[90,2] + -1.531;
   1:  PR[91,3] = PR[90,3] + 35.581;
   1:L PR[91] R[100]mm/sec CNT100;
   1:  PR[91,1] = PR[90,1] + -30.707;
   1:  PR[91,2] = PR[90,2] + -2.463;
   1:  PR[91,3] = PR[90,3] + 35.589;
   1:L PR[91] R[100]mm/sec CNT100;
   1:  PR[91,1] = PR[90,1] + -30.532;
   1:  PR[91,2] = PR[90,2] + -3.373;
   1:  PR[91,3] = PR[90,3] + 35.596;
   1:L PR[91] R[100]mm/sec CNT100;
   1:  PR[91,1] = PR[90,1] + -30.307;
   1:  PR[91,2] = PR[90,2] + -4.271;
   1:  PR[91,3] = PR[90,3] + 35.604;
   1:L PR[91] R[100]mm/sec CNT100;
   1:  PR[91,1] = PR[90,1] + -30.033;
   1:  PR[91,2] = PR[90,2] + -5.161;
   1:  PR[91,3] = PR[90,3] + 35.611;
   1:L PR[91] R[100]mm/sec CNT100;
   1:  PR[91,1] = PR[90,1] + -29.710;
   1:  PR[91,2] = PR[90,2] + -6.044;
   1:  PR[91,3] = PR[90,3] + 35.619;
   1:L PR[91] R[100]mm/sec CNT100;
   1:  PR[91,1] = PR[90,1] + -29.339;
   1:  PR[91,2] = PR[90,2] + -6.923;
   1:  PR[91,3] = PR[90,3] + 35.626;
   1:L PR[91] R[100]mm/sec CNT100;
   1:  PR[91,1] = PR[90,1] + -28.919;
   1:  PR[91,2] = PR[90,2] + -7.792;
   1:  PR[91,3] = PR[90,3] + 35.634;
   1:L PR[91] R[100]mm/sec CNT100;
   1:  PR[91,1] = PR[90,1] + -28.649;
   1:  PR[91,2] = PR[90,2] + -8.290;
   1:  PR[91,3] = PR[90,3] + 35.641;
   1:L PR[91] R[100]mm/sec CNT100;
   1:  PR[91,1] = PR[90,1] + -28.454;
   1:  PR[91,2] = PR[90,2] + -8.644;
   1:  PR[91,3] = PR[90,3] + 35.646;
   1:L PR[91] R[100]mm/sec CNT100;
   1:  PR[91,1] = PR[90,1] + -27.942;
   1:  PR[91,2] = PR[90,2] + -9.478;
   1:  PR[91,3] = PR[90,3] + 35.649;
   1:L PR[91] R[100]mm/sec CNT100;
   1:  PR[91,1] = PR[90,1] + -27.387;
   1:  PR[91,2] = PR[90,2] + -10.286;
   1:  PR[91,3] = PR[90,3] + 35.657;
   1:L PR[91] R[100]mm/sec CNT100;
   1:  PR[91,1] = PR[90,1] + -26.787;
   1:  PR[91,2] = PR[90,2] + -11.065;
   1:  PR[91,3] = PR[90,3] + 35.665;
   1:L PR[91] R[100]mm/sec CNT100;
   1:  PR[91,1] = PR[90,1] + -26.146;
   1:  PR[91,2] = PR[90,2] + -11.815;
   1:  PR[91,3] = PR[90,3] + 35.672;
   1:L PR[91] R[100]mm/sec CNT100;
   1:  PR[91,1] = PR[90,1] + -25.462;
   1:  PR[91,2] = PR[90,2] + -12.533;
   1:  PR[91,3] = PR[90,3] + 35.680;
   1:L PR[91] R[100]mm/sec CNT100;
   1:  PR[91,1] = PR[90,1] + -24.739;
   1:  PR[91,2] = PR[90,2] + -13.218;
   1:  PR[91,3] = PR[90,3] + 35.688;
   1:L PR[91] R[100]mm/sec CNT100;
   1:  PR[91,1] = PR[90,1] + -23.978;
   1:  PR[91,2] = PR[90,2] + -13.868;
   1:  PR[91,3] = PR[90,3] + 35.696;
   1:L PR[91] R[100]mm/sec CNT100;
   1:  PR[91,1] = PR[90,1] + -23.180;
   1:  PR[91,2] = PR[90,2] + -14.483;
   1:  PR[91,3] = PR[90,3] + 35.704;
   1:L PR[91] R[100]mm/sec CNT100;
   1:  PR[91,1] = PR[90,1] + -22.348;
   1:  PR[91,2] = PR[90,2] + -15.059;
   1:  PR[91,3] = PR[90,3] + 35.712;
   1:L PR[91] R[100]mm/sec CNT100;
   1:  PR[91,1] = PR[90,1] + -21.482;
   1:  PR[91,2] = PR[90,2] + -15.597;
   1:  PR[91,3] = PR[90,3] + 35.720;
   1:L PR[91] R[100]mm/sec CNT100;
   1:  PR[91,1] = PR[90,1] + -20.579;
   1:  PR[91,2] = PR[90,2] + -16.097;
   1:  PR[91,3] = PR[90,3] + 35.728;
   1:L PR[91] R[100]mm/sec CNT100;
   1:  PR[91,1] = PR[90,1] + -19.694;
   1:  PR[91,2] = PR[90,2] + -16.534;
   1:  PR[91,3] = PR[90,3] + 35.737;
   1:L PR[91] R[100]mm/sec CNT100;
   1:  PR[91,1] = PR[90,1] + -18.776;
   1:  PR[91,2] = PR[90,2] + -16.933;
   1:  PR[91,3] = PR[90,3] + 35.744;
   1:L PR[91] R[100]mm/sec CNT100;
   1:  PR[91,1] = PR[90,1] + -17.839;
   1:  PR[91,2] = PR[90,2] + -17.287;
   1:  PR[91,3] = PR[90,3] + 35.752;
   1:L PR[91] R[100]mm/sec CNT100;
   1:  PR[91,1] = PR[90,1] + -16.885;
   1:  PR[91,2] = PR[90,2] + -17.596;
   1:  PR[91,3] = PR[90,3] + 35.760;
   1:L PR[91] R[100]mm/sec CNT100;
   1:  PR[91,1] = PR[90,1] + -15.915;
   1:  PR[91,2] = PR[90,2] + -17.858;
   1:  PR[91,3] = PR[90,3] + 35.768;
   1:L PR[91] R[100]mm/sec CNT100;
   1:  PR[91,1] = PR[90,1] + -14.934;
   1:  PR[91,2] = PR[90,2] + -18.073;
   1:  PR[91,3] = PR[90,3] + 35.776;
   1:L PR[91] R[100]mm/sec CNT100;
   1:  PR[91,1] = PR[90,1] + -13.942;
   1:  PR[91,2] = PR[90,2] + -18.240;
   1:  PR[91,3] = PR[90,3] + 35.784;
   1:L PR[91] R[100]mm/sec CNT100;
   1:  PR[91,1] = PR[90,1] + -12.943;
   1:  PR[91,2] = PR[90,2] + -18.360;
   1:  PR[91,3] = PR[90,3] + 35.792;
   1:L PR[91] R[100]mm/sec CNT100;
   1:  PR[91,1] = PR[90,1] + -11.941;
   1:  PR[91,2] = PR[90,2] + -18.431;
   1:  PR[91,3] = PR[90,3] + 35.800;
   1:L PR[91] R[100]mm/sec CNT100;
   1:  PR[91,1] = PR[90,1] + -10.935;
   1:  PR[91,2] = PR[90,2] + -18.453;
   1:  PR[91,3] = PR[90,3] + 35.808;
   1:L PR[91] R[100]mm/sec CNT100;
   1:  PR[91,1] = PR[90,1] + -9.930;
   1:  PR[91,2] = PR[90,2] + -18.427;
   1:  PR[91,3] = PR[90,3] + 35.816;
   1:L PR[91] R[100]mm/sec CNT100;
   1:  PR[91,1] = PR[90,1] + -8.928;
   1:  PR[91,2] = PR[90,2] + -18.353;
   1:  PR[91,3] = PR[90,3] + 35.824;
   1:L PR[91] R[100]mm/sec CNT100;
   1:  PR[91,1] = PR[90,1] + -7.932;
   1:  PR[91,2] = PR[90,2] + -18.230;
   1:  PR[91,3] = PR[90,3] + 35.832;
   1:L PR[91] R[100]mm/sec CNT100;
   1:  PR[91,1] = PR[90,1] + -6.943;
   1:  PR[91,2] = PR[90,2] + -18.059;
   1:  PR[91,3] = PR[90,3] + 35.840;
   1:L PR[91] R[100]mm/sec CNT100;
   1:  PR[91,1] = PR[90,1] + -5.965;
   1:  PR[91,2] = PR[90,2] + -17.840;
   1:  PR[91,3] = PR[90,3] + 35.848;
   1:L PR[91] R[100]mm/sec CNT100;
   1:  PR[91,1] = PR[90,1] + -4.979;
   1:  PR[91,2] = PR[90,2] + -17.568;
   1:  PR[91,3] = PR[90,3] + 35.856;
   1:L PR[91] R[100]mm/sec CNT100;
   1:  PR[91,1] = PR[90,1] + -4.045;
   1:  PR[91,2] = PR[90,2] + -17.260;
   1:  PR[91,3] = PR[90,3] + 35.864;
   1:L PR[91] R[100]mm/sec CNT100;
   1:  PR[91,1] = PR[90,1] + -3.109;
   1:  PR[91,2] = PR[90,2] + -16.900;
   1:  PR[91,3] = PR[90,3] + 35.872;
   1:L PR[91] R[100]mm/sec CNT100;
   1:  PR[91,1] = PR[90,1] + -2.194;
   1:  PR[91,2] = PR[90,2] + -16.495;
   1:  PR[91,3] = PR[90,3] + 35.880;
   1:L PR[91] R[100]mm/sec CNT100;
   1:  PR[91,1] = PR[90,1] + -1.475;
   1:  PR[91,2] = PR[90,2] + -16.135;
   1:  PR[91,3] = PR[90,3] + 35.888;
   1:L PR[91] R[100]mm/sec CNT100;
   1:  PR[91,1] = PR[90,1] + -1.050;
   1:  PR[91,2] = PR[90,2] + -15.956;
   1:  PR[91,3] = PR[90,3] + 35.895;
   1:L PR[91] R[100]mm/sec CNT100;
   1:  PR[91,1] = PR[90,1] + -0.574;
   1:  PR[91,2] = PR[90,2] + -15.842;
   1:  PR[91,3] = PR[90,3] + 35.898;
   1:L PR[91] R[100]mm/sec CNT100;
   1:  PR[91,1] = PR[90,1] + -0.086;
   1:  PR[91,2] = PR[90,2] + -15.807;
   1:  PR[91,3] = PR[90,3] + 35.902;
   1:L PR[91] R[100]mm/sec CNT100;
   1:  PR[91,1] = PR[90,1] + 0.406;
   1:  PR[91,2] = PR[90,2] + -15.852;
   1:  PR[91,3] = PR[90,3] + 35.906;
   1:L PR[91] R[100]mm/sec CNT100;
   1:  PR[91] = PR[90];
   1:  PR[91,1] = PR[90,1] + 0.951;
   1:  PR[91,2] = PR[90,2] + -16.464;
   1:  PR[91,3] = PR[90,3] + 37.240;
   1:L PR[91] R[100]mm/sec CNT100;
   1:  PR[91,1] = PR[90,1] + 2.423;
   1:  PR[91,2] = PR[90,2] + -17.122;
   1:  PR[91,3] = PR[90,3] + 35.914;
   1:L PR[91] R[100]mm/sec CNT100;
   1:  PR[91,1] = PR[90,1] + 3.362;
   1:  PR[91,2] = PR[90,2] + -17.476;
   1:  PR[91,3] = PR[90,3] + 35.927;
   1:L PR[91] R[100]mm/sec CNT100;
   1:  PR[91,1] = PR[90,1] + 4.322;
   1:  PR[91,2] = PR[90,2] + -17.785;
   1:  PR[91,3] = PR[90,3] + 35.935;
   1:L PR[91] R[100]mm/sec CNT100;
   1:  PR[91,1] = PR[90,1] + 5.298;
   1:  PR[91,2] = PR[90,2] + -18.047;
   1:  PR[91,3] = PR[90,3] + 35.943;
   1:L PR[91] R[100]mm/sec CNT100;
   1:  PR[91,1] = PR[90,1] + 5.906;
   1:  PR[91,2] = PR[90,2] + -18.182;
   1:  PR[91,3] = PR[90,3] + 35.951;
   1:L PR[91] R[100]mm/sec CNT100;
   1:  PR[91,1] = PR[90,1] + 6.282;
   1:  PR[91,2] = PR[90,2] + -18.261;
   1:  PR[91,3] = PR[90,3] + 35.956;
   1:L PR[91] R[100]mm/sec CNT100;
   1:  PR[91,1] = PR[90,1] + 7.282;
   1:  PR[91,2] = PR[90,2] + -18.426;
   1:  PR[91,3] = PR[90,3] + 35.959;
   1:L PR[91] R[100]mm/sec CNT100;
   1:  PR[91,1] = PR[90,1] + 8.287;
   1:  PR[91,2] = PR[90,2] + -18.543;
   1:  PR[91,3] = PR[90,3] + 35.967;
   1:L PR[91] R[100]mm/sec CNT100;
   1:  PR[91,1] = PR[90,1] + 9.092;
   1:  PR[91,2] = PR[90,2] + -18.599;
   1:  PR[91,3] = PR[90,3] + 35.975;
   1:L PR[91] R[100]mm/sec CNT100;
   1:  PR[91,1] = PR[90,1] + 10.310;
   1:  PR[91,2] = PR[90,2] + -18.628;
   1:  PR[91,3] = PR[90,3] + 35.982;
   1:L PR[91] R[100]mm/sec CNT100;
   1:  PR[91,1] = PR[90,1] + 11.320;
   1:  PR[91,2] = PR[90,2] + -18.598;
   1:  PR[91,3] = PR[90,3] + 35.992;
   1:L PR[91] R[100]mm/sec CNT100;
   1:  PR[91,1] = PR[90,1] + 12.329;
   1:  PR[91,2] = PR[90,2] + -18.518;
   1:  PR[91,3] = PR[90,3] + 36.000;
   1:L PR[91] R[100]mm/sec CNT100;
   1:  PR[91,1] = PR[90,1] + 13.331;
   1:  PR[91,2] = PR[90,2] + -18.392;
   1:  PR[91,3] = PR[90,3] + 36.008;
   1:L PR[91] R[100]mm/sec CNT100;
   1:  PR[91,1] = PR[90,1] + 14.324;
   1:  PR[91,2] = PR[90,2] + -18.218;
   1:  PR[91,3] = PR[90,3] + 36.016;
   1:L PR[91] R[100]mm/sec CNT100;
   1:  PR[91,1] = PR[90,1] + 15.307;
   1:  PR[91,2] = PR[90,2] + -17.996;
   1:  PR[91,3] = PR[90,3] + 36.024;
   1:L PR[91] R[100]mm/sec CNT100;
   1:  PR[91,1] = PR[90,1] + 16.278;
   1:  PR[91,2] = PR[90,2] + -17.726;
   1:  PR[91,3] = PR[90,3] + 36.032;
   1:L PR[91] R[100]mm/sec CNT100;
   1:  PR[91,1] = PR[90,1] + 17.233;
   1:  PR[91,2] = PR[90,2] + -17.411;
   1:  PR[91,3] = PR[90,3] + 36.040;
   1:L PR[91] R[100]mm/sec CNT100;
   1:  PR[91,1] = PR[90,1] + 18.172;
   1:  PR[91,2] = PR[90,2] + -17.051;
   1:  PR[91,3] = PR[90,3] + 36.048;
   1:L PR[91] R[100]mm/sec CNT100;
   1:  PR[91,1] = PR[90,1] + 19.091;
   1:  PR[91,2] = PR[90,2] + -16.646;
   1:  PR[91,3] = PR[90,3] + 36.056;
   1:L PR[91] R[100]mm/sec CNT100;
   1:  PR[91,1] = PR[90,1] + 19.989;
   1:  PR[91,2] = PR[90,2] + -16.198;
   1:  PR[91,3] = PR[90,3] + 36.065;
   1:L PR[91] R[100]mm/sec CNT100;
   1:  PR[91,1] = PR[90,1] + 20.445;
   1:  PR[91,2] = PR[90,2] + -15.945;
   1:  PR[91,3] = PR[90,3] + 36.073;
   1:L PR[91] R[100]mm/sec CNT100;
   1:  PR[91,1] = PR[90,1] + 20.858;
   1:  PR[91,2] = PR[90,2] + -15.710;
   1:  PR[91,3] = PR[90,3] + 36.077;
   1:L PR[91] R[100]mm/sec CNT100;
   1:  PR[91,1] = PR[90,1] + 21.704;
   1:  PR[91,2] = PR[90,2] + -15.179;
   1:  PR[91,3] = PR[90,3] + 36.081;
   1:L PR[91] R[100]mm/sec CNT100;
   1:  PR[91,1] = PR[90,1] + 22.520;
   1:  PR[91,2] = PR[90,2] + -14.609;
   1:  PR[91,3] = PR[90,3] + 36.089;
   1:L PR[91] R[100]mm/sec CNT100;
   1:  PR[91,1] = PR[90,1] + 23.306;
   1:  PR[91,2] = PR[90,2] + -14.000;
   1:  PR[91,3] = PR[90,3] + 36.097;
   1:L PR[91] R[100]mm/sec CNT100;
   1:  PR[91,1] = PR[90,1] + 24.057;
   1:  PR[91,2] = PR[90,2] + -13.354;
   1:  PR[91,3] = PR[90,3] + 36.105;
   1:L PR[91] R[100]mm/sec CNT100;
   1:  PR[91,1] = PR[90,1] + 24.774;
   1:  PR[91,2] = PR[90,2] + -12.672;
   1:  PR[91,3] = PR[90,3] + 36.113;
   1:L PR[91] R[100]mm/sec CNT100;
   1:  PR[91,1] = PR[90,1] + 25.454;
   1:  PR[91,2] = PR[90,2] + -11.955;
   1:  PR[91,3] = PR[90,3] + 36.120;
   1:L PR[91] R[100]mm/sec CNT100;
   1:  PR[91,1] = PR[90,1] + 26.095;
   1:  PR[91,2] = PR[90,2] + -11.204;
   1:  PR[91,3] = PR[90,3] + 36.128;
   1:L PR[91] R[100]mm/sec CNT100;
   1:  PR[91,1] = PR[90,1] + 26.696;
   1:  PR[91,2] = PR[90,2] + -10.422;
   1:  PR[91,3] = PR[90,3] + 36.136;
   1:L PR[91] R[100]mm/sec CNT100;
   1:  PR[91,1] = PR[90,1] + 27.257;
   1:  PR[91,2] = PR[90,2] + -9.609;
   1:  PR[91,3] = PR[90,3] + 36.144;
   1:L PR[91] R[100]mm/sec CNT100;
   1:  PR[91,1] = PR[90,1] + 27.778;
   1:  PR[91,2] = PR[90,2] + -8.767;
   1:  PR[91,3] = PR[90,3] + 36.152;
   1:L PR[91] R[100]mm/sec CNT100;
   1:  PR[91,1] = PR[90,1] + 28.253;
   1:  PR[91,2] = PR[90,2] + -7.906;
   1:  PR[91,3] = PR[90,3] + 36.160;
   1:L PR[91] R[100]mm/sec CNT100;
   1:  PR[91,1] = PR[90,1] + 28.680;
   1:  PR[91,2] = PR[90,2] + -7.031;
   1:  PR[91,3] = PR[90,3] + 36.168;
   1:L PR[91] R[100]mm/sec CNT100;
   1:  PR[91,1] = PR[90,1] + 29.058;
   1:  PR[91,2] = PR[90,2] + -6.147;
   1:  PR[91,3] = PR[90,3] + 36.176;
   1:L PR[91] R[100]mm/sec CNT100;
   1:  PR[91,1] = PR[90,1] + 29.387;
   1:  PR[91,2] = PR[90,2] + -5.255;
   1:  PR[91,3] = PR[90,3] + 36.184;
   1:L PR[91] R[100]mm/sec CNT100;
   1:  PR[91,1] = PR[90,1] + 29.666;
   1:  PR[91,2] = PR[90,2] + -4.354;
   1:  PR[91,3] = PR[90,3] + 36.191;
   1:L PR[91] R[100]mm/sec CNT100;
   1:  PR[91,1] = PR[90,1] + 29.894;
   1:  PR[91,2] = PR[90,2] + -3.442;
   1:  PR[91,3] = PR[90,3] + 36.199;
   1:L PR[91] R[100]mm/sec CNT100;
   1:  PR[91,1] = PR[90,1] + 30.073;
   1:  PR[91,2] = PR[90,2] + -2.512;
   1:  PR[91,3] = PR[90,3] + 36.206;
   1:L PR[91] R[100]mm/sec CNT100;
   1:  PR[91,1] = PR[90,1] + 30.200;
   1:  PR[91,2] = PR[90,2] + -1.561;
   1:  PR[91,3] = PR[90,3] + 36.214;
   1:L PR[91] R[100]mm/sec CNT100;
   1:  PR[91,1] = PR[90,1] + 30.277;
   1:  PR[91,2] = PR[90,2] + -0.583;
   1:  PR[91,3] = PR[90,3] + 36.222;
   1:L PR[91] R[100]mm/sec CNT100;
   1:  PR[91,1] = PR[90,1] + 30.302;
   1:  PR[91,2] = PR[90,2] + 0.428;
   1:  PR[91,3] = PR[90,3] + 36.229;
   1:L PR[91] R[100]mm/sec CNT100;
   1:  PR[91,1] = PR[90,1] + 30.277;
   1:  PR[91,2] = PR[90,2] + 1.438;
   1:  PR[91,3] = PR[90,3] + 36.238;
   1:L PR[91] R[100]mm/sec CNT100;
   1:  PR[91,1] = PR[90,1] + 30.200;
   1:  PR[91,2] = PR[90,2] + 2.417;
   1:  PR[91,3] = PR[90,3] + 36.246;
   1:L PR[91] R[100]mm/sec CNT100;
   1:  PR[91,1] = PR[90,1] + 30.073;
   1:  PR[91,2] = PR[90,2] + 3.368;
   1:  PR[91,3] = PR[90,3] + 36.254;
   1:L PR[91] R[100]mm/sec CNT100;
   1:  PR[91,1] = PR[90,1] + 29.894;
   1:  PR[91,2] = PR[90,2] + 4.297;
   1:  PR[91,3] = PR[90,3] + 36.261;
   1:L PR[91] R[100]mm/sec CNT100;
   1:  PR[91,1] = PR[90,1] + 29.666;
   1:  PR[91,2] = PR[90,2] + 5.209;
   1:  PR[91,3] = PR[90,3] + 36.269;
   1:L PR[91] R[100]mm/sec CNT100;
   1:  PR[91,1] = PR[90,1] + 29.387;
   1:  PR[91,2] = PR[90,2] + 6.110;
   1:  PR[91,3] = PR[90,3] + 36.276;
   1:L PR[91] R[100]mm/sec CNT100;
   1:  PR[91,1] = PR[90,1] + 29.058;
   1:  PR[91,2] = PR[90,2] + 7.002;
   1:  PR[91,3] = PR[90,3] + 36.284;
   1:L PR[91] R[100]mm/sec CNT100;
   1:  PR[91,1] = PR[90,1] + 28.680;
   1:  PR[91,2] = PR[90,2] + 7.886;
   1:  PR[91,3] = PR[90,3] + 36.292;
   1:L PR[91] R[100]mm/sec CNT100;
   1:  PR[91,1] = PR[90,1] + 28.253;
   1:  PR[91,2] = PR[90,2] + 8.761;
   1:  PR[91,3] = PR[90,3] + 36.299;
   1:L PR[91] R[100]mm/sec CNT100;
   1:  PR[91,1] = PR[90,1] + 27.778;
   1:  PR[91,2] = PR[90,2] + 9.622;
   1:  PR[91,3] = PR[90,3] + 36.307;
   1:L PR[91] R[100]mm/sec CNT100;
   1:  PR[91,1] = PR[90,1] + 27.252;
   1:  PR[91,2] = PR[90,2] + 10.471;
   1:  PR[91,3] = PR[90,3] + 36.315;
   1:L PR[91] R[100]mm/sec CNT100;
   1:  PR[91,1] = PR[90,1] + 26.696;
   1:  PR[91,2] = PR[90,2] + 11.277;
   1:  PR[91,3] = PR[90,3] + 36.323;
   1:L PR[91] R[100]mm/sec CNT100;
   1:  PR[91,1] = PR[90,1] + 26.095;
   1:  PR[91,2] = PR[90,2] + 12.059;
   1:  PR[91,3] = PR[90,3] + 36.331;
   1:L PR[91] R[100]mm/sec CNT100;
   1:  PR[91,1] = PR[90,1] + 25.454;
   1:  PR[91,2] = PR[90,2] + 12.810;
   1:  PR[91,3] = PR[90,3] + 36.339;
   1:L PR[91] R[100]mm/sec CNT100;
   1:  PR[91,1] = PR[90,1] + 24.776;
   1:  PR[91,2] = PR[90,2] + 13.526;
   1:  PR[91,3] = PR[90,3] + 36.347;
   1:L PR[91] R[100]mm/sec CNT100;
   1:  PR[91,1] = PR[90,1] + 23.877;
   1:  PR[91,2] = PR[90,2] + 14.367;
   1:  PR[91,3] = PR[90,3] + 36.355;
   1:L PR[91] R[100]mm/sec CNT100;
   1:  PR[91,1] = PR[90,1] + 23.306;
   1:  PR[91,2] = PR[90,2] + 14.855;
   1:  PR[91,3] = PR[90,3] + 36.365;
   1:L PR[91] R[100]mm/sec CNT100;
   1:  PR[91,1] = PR[90,1] + 22.520;
   1:  PR[91,2] = PR[90,2] + 15.464;
   1:  PR[91,3] = PR[90,3] + 36.371;
   1:L PR[91] R[100]mm/sec CNT100;
   1:  PR[91,1] = PR[90,1] + 21.704;
   1:  PR[91,2] = PR[90,2] + 16.034;
   1:  PR[91,3] = PR[90,3] + 36.379;
   1:L PR[91] R[100]mm/sec CNT100;
   1:  PR[91,1] = PR[90,1] + 20.859;
   1:  PR[91,2] = PR[90,2] + 16.565;
   1:  PR[91,3] = PR[90,3] + 36.387;
   1:L PR[91] R[100]mm/sec CNT100;
   1:  PR[91,1] = PR[90,1] + 19.985;
   1:  PR[91,2] = PR[90,2] + 17.055;
   1:  PR[91,3] = PR[90,3] + 36.395;
   1:L PR[91] R[100]mm/sec CNT100;
   1:  PR[91,1] = PR[90,1] + 19.503;
   1:  PR[91,2] = PR[90,2] + 17.299;
   1:  PR[91,3] = PR[90,3] + 36.403;
   1:L PR[91] R[100]mm/sec CNT100;
   1:  PR[91,1] = PR[90,1] + 19.092;
   1:  PR[91,2] = PR[90,2] + 17.501;
   1:  PR[91,3] = PR[90,3] + 36.407;
   1:L PR[91] R[100]mm/sec CNT100;
   1:  PR[91,1] = PR[90,1] + 18.171;
   1:  PR[91,2] = PR[90,2] + 17.906;
   1:  PR[91,3] = PR[90,3] + 36.411;
   1:L PR[91] R[100]mm/sec CNT100;
   1:  PR[91,1] = PR[90,1] + 17.232;
   1:  PR[91,2] = PR[90,2] + 18.267;
   1:  PR[91,3] = PR[90,3] + 36.419;
   1:L PR[91] R[100]mm/sec CNT100;
   1:  PR[91,1] = PR[90,1] + 16.276;
   1:  PR[91,2] = PR[90,2] + 18.582;
   1:  PR[91,3] = PR[90,3] + 36.427;
   1:L PR[91] R[100]mm/sec CNT100;
   1:  PR[91,1] = PR[90,1] + 15.305;
   1:  PR[91,2] = PR[90,2] + 18.851;
   1:  PR[91,3] = PR[90,3] + 36.435;
   1:L PR[91] R[100]mm/sec CNT100;
   1:  PR[91,1] = PR[90,1] + 14.322;
   1:  PR[91,2] = PR[90,2] + 19.073;
   1:  PR[91,3] = PR[90,3] + 36.443;
   1:L PR[91] R[100]mm/sec CNT100;
   1:  PR[91,1] = PR[90,1] + 13.329;
   1:  PR[91,2] = PR[90,2] + 19.247;
   1:  PR[91,3] = PR[90,3] + 36.451;
   1:L PR[91] R[100]mm/sec CNT100;
   1:  PR[91,1] = PR[90,1] + 12.324;
   1:  PR[91,2] = PR[90,2] + 19.374;
   1:  PR[91,3] = PR[90,3] + 36.459;
   1:L PR[91] R[100]mm/sec CNT100;
   1:  PR[91,1] = PR[90,1] + 11.317;
   1:  PR[91,2] = PR[90,2] + 19.453;
   1:  PR[91,3] = PR[90,3] + 36.467;
   1:L PR[91] R[100]mm/sec CNT100;
   1:  PR[91,1] = PR[90,1] + 10.308;
   1:  PR[91,2] = PR[90,2] + 19.484;
   1:  PR[91,3] = PR[90,3] + 36.475;
   1:L PR[91] R[100]mm/sec CNT100;
   1:  PR[91,1] = PR[90,1] + 9.090;
   1:  PR[91,2] = PR[90,2] + 19.454;
   1:  PR[91,3] = PR[90,3] + 36.484;
   1:L PR[91] R[100]mm/sec CNT100;
   1:  PR[91,1] = PR[90,1] + 8.285;
   1:  PR[91,2] = PR[90,2] + 19.398;
   1:  PR[91,3] = PR[90,3] + 36.493;
   1:L PR[91] R[100]mm/sec CNT100;
   1:  PR[91,1] = PR[90,1] + 7.279;
   1:  PR[91,2] = PR[90,2] + 19.281;
   1:  PR[91,3] = PR[90,3] + 36.500;
   1:L PR[91] R[100]mm/sec CNT100;
   1:  PR[91,1] = PR[90,1] + 6.282;
   1:  PR[91,2] = PR[90,2] + 19.116;
   1:  PR[91,3] = PR[90,3] + 36.508;
   1:L PR[91] R[100]mm/sec CNT100;
   1:  PR[91,1] = PR[90,1] + 5.295;
   1:  PR[91,2] = PR[90,2] + 18.902;
   1:  PR[91,3] = PR[90,3] + 36.516;
   1:L PR[91] R[100]mm/sec CNT100;
   1:  PR[91,1] = PR[90,1] + 4.320;
   1:  PR[91,2] = PR[90,2] + 18.639;
   1:  PR[91,3] = PR[90,3] + 36.524;
   1:L PR[91] R[100]mm/sec CNT100;
   1:  PR[91,1] = PR[90,1] + 3.360;
   1:  PR[91,2] = PR[90,2] + 18.330;
   1:  PR[91,3] = PR[90,3] + 36.532;
   1:L PR[91] R[100]mm/sec CNT100;
   1:  PR[91,1] = PR[90,1] + 2.418;
   1:  PR[91,2] = PR[90,2] + 17.975;
   1:  PR[91,3] = PR[90,3] + 36.540;
   1:L PR[91] R[100]mm/sec CNT100;
   1:  PR[91,1] = PR[90,1] + 1.492;
   1:  PR[91,2] = PR[90,2] + 17.573;
   1:  PR[91,3] = PR[90,3] + 36.548;
   1:L PR[91] R[100]mm/sec CNT100;
   1:  PR[91,1] = PR[90,1] + 0.957;
   1:  PR[91,2] = PR[90,2] + 17.321;
   1:  PR[91,3] = PR[90,3] + 36.557;
   1:L PR[91] R[100]mm/sec CNT100;
   1:  PR[91,1] = PR[90,1] + 0.487;
   1:  PR[91,2] = PR[90,2] + 17.182;
   1:  PR[91,3] = PR[90,3] + 36.561;
   1:L PR[91] R[100]mm/sec CNT100;
   1:  PR[91,1] = PR[90,1] + -0.002;
   1:  PR[91,2] = PR[90,2] + 17.121;
   1:  PR[91,3] = PR[90,3] + 36.565;
   1:L PR[91] R[100]mm/sec CNT100;
   1:  PR[91,1] = PR[90,1] + -0.493;
   1:  PR[91,2] = PR[90,2] + 17.142;
   1:  PR[91,3] = PR[90,3] + 36.569;
   1:L PR[91] R[100]mm/sec CNT100;
   1:  PR[91,1] = PR[90,1] + -0.972;
   1:  PR[91,2] = PR[90,2] + 17.244;
   1:  PR[91,3] = PR[90,3] + 36.573;
   1:L PR[91] R[100]mm/sec CNT100;
   1:  PR[91,1] = PR[90,1] + -1.401;
   1:  PR[91,2] = PR[90,2] + 17.412;
   1:  PR[91,3] = PR[90,3] + 36.577;
   1:L PR[91] R[100]mm/sec CNT100;
   1:  PR[91,1] = PR[90,1] + -2.099;
   1:  PR[91,2] = PR[90,2] + 17.736;
   1:  PR[91,3] = PR[90,3] + 36.581;
   1:L PR[91] R[100]mm/sec CNT100;
   1:  PR[91,1] = PR[90,1] + -2.658;
   1:  PR[91,2] = PR[90,2] + 17.976;
   1:  PR[91,3] = PR[90,3] + 36.587;
   1:L PR[91] R[100]mm/sec CNT100;
   1:  PR[91,1] = PR[90,1] + -3.602;
   1:  PR[91,2] = PR[90,2] + 18.333;
   1:  PR[91,3] = PR[90,3] + 36.592;
   1:L PR[91] R[100]mm/sec CNT100;
   1:  PR[91,1] = PR[90,1] + -4.561;
   1:  PR[91,2] = PR[90,2] + 18.642;
   1:  PR[91,3] = PR[90,3] + 36.600;
   1:L PR[91] R[100]mm/sec CNT100;
   1:  PR[91,1] = PR[90,1] + -5.537;
   1:  PR[91,2] = PR[90,2] + 18.904;
   1:  PR[91,3] = PR[90,3] + 36.608;
   1:L PR[91] R[100]mm/sec CNT100;
   1:  PR[91,1] = PR[90,1] + -6.145;
   1:  PR[91,2] = PR[90,2] + 19.038;
   1:  PR[91,3] = PR[90,3] + 36.616;
   1:L PR[91] R[100]mm/sec CNT100;
   1:  PR[91,1] = PR[90,1] + -6.521;
   1:  PR[91,2] = PR[90,2] + 19.116;
   1:  PR[91,3] = PR[90,3] + 36.621;
   1:L PR[91] R[100]mm/sec CNT100;
   1:  PR[91,1] = PR[90,1] + -7.521;
   1:  PR[91,2] = PR[90,2] + 19.282;
   1:  PR[91,3] = PR[90,3] + 36.624;
   1:L PR[91] R[100]mm/sec CNT100;
   1:  PR[91,1] = PR[90,1] + -8.526;
   1:  PR[91,2] = PR[90,2] + 19.398;
   1:  PR[91,3] = PR[90,3] + 36.632;
   1:L PR[91] R[100]mm/sec CNT100;
   1:  PR[91,1] = PR[90,1] + -9.332;
   1:  PR[91,2] = PR[90,2] + 19.453;
   1:  PR[91,3] = PR[90,3] + 36.640;
   1:L PR[91] R[100]mm/sec CNT100;
   1:  PR[91,1] = PR[90,1] + -10.549;
   1:  PR[91,2] = PR[90,2] + 19.483;
   1:  PR[91,3] = PR[90,3] + 36.647;
   1:L PR[91] R[100]mm/sec CNT100;
   1:  PR[91,1] = PR[90,1] + -11.559;
   1:  PR[91,2] = PR[90,2] + 19.453;
   1:  PR[91,3] = PR[90,3] + 36.657;
   1:L PR[91] R[100]mm/sec CNT100;
   1:  PR[91,1] = PR[90,1] + -12.568;
   1:  PR[91,2] = PR[90,2] + 19.373;
   1:  PR[91,3] = PR[90,3] + 36.665;
   1:L PR[91] R[100]mm/sec CNT100;
   1:  PR[91,1] = PR[90,1] + -13.570;
   1:  PR[91,2] = PR[90,2] + 19.247;
   1:  PR[91,3] = PR[90,3] + 36.673;
   1:L PR[91] R[100]mm/sec CNT100;
   1:  PR[91,1] = PR[90,1] + -14.564;
   1:  PR[91,2] = PR[90,2] + 19.072;
   1:  PR[91,3] = PR[90,3] + 36.681;
   1:L PR[91] R[100]mm/sec CNT100;
   1:  PR[91,1] = PR[90,1] + -15.547;
   1:  PR[91,2] = PR[90,2] + 18.851;
   1:  PR[91,3] = PR[90,3] + 36.689;
   1:L PR[91] R[100]mm/sec CNT100;
   1:  PR[91,1] = PR[90,1] + -16.518;
   1:  PR[91,2] = PR[90,2] + 18.582;
   1:  PR[91,3] = PR[90,3] + 36.697;
   1:L PR[91] R[100]mm/sec CNT100;
   1:  PR[91,1] = PR[90,1] + -17.474;
   1:  PR[91,2] = PR[90,2] + 18.267;
   1:  PR[91,3] = PR[90,3] + 36.705;
   1:L PR[91] R[100]mm/sec CNT100;
   1:  PR[91,1] = PR[90,1] + -18.412;
   1:  PR[91,2] = PR[90,2] + 17.907;
   1:  PR[91,3] = PR[90,3] + 36.713;
   1:L PR[91] R[100]mm/sec CNT100;
   1:  PR[91,1] = PR[90,1] + -19.330;
   1:  PR[91,2] = PR[90,2] + 17.501;
   1:  PR[91,3] = PR[90,3] + 36.721;
   1:L PR[91] R[100]mm/sec CNT100;
   1:  PR[91,1] = PR[90,1] + -20.227;
   1:  PR[91,2] = PR[90,2] + 17.052;
   1:  PR[91,3] = PR[90,3] + 36.730;
   1:L PR[91] R[100]mm/sec CNT100;
   1:  PR[91,1] = PR[90,1] + -21.100;
   1:  PR[91,2] = PR[90,2] + 16.561;
   1:  PR[91,3] = PR[90,3] + 36.738;
   1:L PR[91] R[100]mm/sec CNT100;
   1:  PR[91,1] = PR[90,1] + -21.597;
   1:  PR[91,2] = PR[90,2] + 16.252;
   1:  PR[91,3] = PR[90,3] + 36.746;
   1:L PR[91] R[100]mm/sec CNT100;
   1:  PR[91,1] = PR[90,1] + -21.943;
   1:  PR[91,2] = PR[90,2] + 16.031;
   1:  PR[91,3] = PR[90,3] + 36.750;
   1:L PR[91] R[100]mm/sec CNT100;
   1:  PR[91,1] = PR[90,1] + -22.761;
   1:  PR[91,2] = PR[90,2] + 15.460;
   1:  PR[91,3] = PR[90,3] + 36.754;
   1:L PR[91] R[100]mm/sec CNT100;
   1:  PR[91,1] = PR[90,1] + -23.546;
   1:  PR[91,2] = PR[90,2] + 14.851;
   1:  PR[91,3] = PR[90,3] + 36.762;
   1:L PR[91] R[100]mm/sec CNT100;
   1:  PR[91,1] = PR[90,1] + -24.298;
   1:  PR[91,2] = PR[90,2] + 14.206;
   1:  PR[91,3] = PR[90,3] + 36.770;
   1:L PR[91] R[100]mm/sec CNT100;
   1:  PR[91,1] = PR[90,1] + -25.015;
   1:  PR[91,2] = PR[90,2] + 13.525;
   1:  PR[91,3] = PR[90,3] + 36.778;
   1:L PR[91] R[100]mm/sec CNT100;
   1:  PR[91,1] = PR[90,1] + -25.694;
   1:  PR[91,2] = PR[90,2] + 12.811;
   1:  PR[91,3] = PR[90,3] + 36.785;
   1:L PR[91] R[100]mm/sec CNT100;
   1:  PR[91,1] = PR[90,1] + -26.336;
   1:  PR[91,2] = PR[90,2] + 12.063;
   1:  PR[91,3] = PR[90,3] + 36.793;
   1:L PR[91] R[100]mm/sec CNT100;
   1:  PR[91,1] = PR[90,1] + -26.936;
   1:  PR[91,2] = PR[90,2] + 11.283;
   1:  PR[91,3] = PR[90,3] + 36.801;
   1:L PR[91] R[100]mm/sec CNT100;
   1:  PR[91,1] = PR[90,1] + -27.496;
   1:  PR[91,2] = PR[90,2] + 10.472;
   1:  PR[91,3] = PR[90,3] + 36.809;
   1:L PR[91] R[100]mm/sec CNT100;
   1:  PR[91,1] = PR[90,1] + -28.017;
   1:  PR[91,2] = PR[90,2] + 9.629;
   1:  PR[91,3] = PR[90,3] + 36.817;
   1:L PR[91] R[100]mm/sec CNT100;
   1:  PR[91,1] = PR[90,1] + -28.491;
   1:  PR[91,2] = PR[90,2] + 8.764;
   1:  PR[91,3] = PR[90,3] + 36.825;
   1:L PR[91] R[100]mm/sec CNT100;
   1:  PR[91,1] = PR[90,1] + -28.918;
   1:  PR[91,2] = PR[90,2] + 7.884;
   1:  PR[91,3] = PR[90,3] + 36.833;
   1:L PR[91] R[100]mm/sec CNT100;
   1:  PR[91,1] = PR[90,1] + -29.296;
   1:  PR[91,2] = PR[90,2] + 6.993;
   1:  PR[91,3] = PR[90,3] + 36.841;
   1:L PR[91] R[100]mm/sec CNT100;
   1:  PR[91,1] = PR[90,1] + -29.625;
   1:  PR[91,2] = PR[90,2] + 6.096;
   1:  PR[91,3] = PR[90,3] + 36.849;
   1:L PR[91] R[100]mm/sec CNT100;
   1:  PR[91,1] = PR[90,1] + -29.905;
   1:  PR[91,2] = PR[90,2] + 5.192;
   1:  PR[91,3] = PR[90,3] + 36.856;
   1:L PR[91] R[100]mm/sec CNT100;
   1:  PR[91,1] = PR[90,1] + -30.133;
   1:  PR[91,2] = PR[90,2] + 4.281;
   1:  PR[91,3] = PR[90,3] + 36.864;
   1:L PR[91] R[100]mm/sec CNT100;
   1:  PR[91,1] = PR[90,1] + -30.311;
   1:  PR[91,2] = PR[90,2] + 3.356;
   1:  PR[91,3] = PR[90,3] + 36.871;
   1:L PR[91] R[100]mm/sec CNT100;
   1:  PR[91,1] = PR[90,1] + -30.439;
   1:  PR[91,2] = PR[90,2] + 2.410;
   1:  PR[91,3] = PR[90,3] + 36.879;
   1:L PR[91] R[100]mm/sec CNT100;
   1:  PR[91,1] = PR[90,1] + -30.516;
   1:  PR[91,2] = PR[90,2] + 1.437;
   1:  PR[91,3] = PR[90,3] + 36.887;
   1:L PR[91] R[100]mm/sec CNT100;
   1:  PR[91,1] = PR[90,1] + -30.540;
   1:  PR[91,2] = PR[90,2] + 0.428;
   1:  PR[91,3] = PR[90,3] + 36.894;
   1:L PR[91] R[100]mm/sec CNT100;
   1:  PR[91,1] = PR[90,1] + -30.516;
   1:  PR[91,2] = PR[90,2] + -0.582;
   1:  PR[91,3] = PR[90,3] + 36.903;
   1:L PR[91] R[100]mm/sec CNT100;
   1:  PR[91,1] = PR[90,1] + -30.439;
   1:  PR[91,2] = PR[90,2] + -1.555;
   1:  PR[91,3] = PR[90,3] + 36.911;
   1:L PR[91] R[100]mm/sec CNT100;
   1:  PR[91,1] = PR[90,1] + -30.311;
   1:  PR[91,2] = PR[90,2] + -2.501;
   1:  PR[91,3] = PR[90,3] + 36.919;
   1:L PR[91] R[100]mm/sec CNT100;
   1:  PR[91,1] = PR[90,1] + -30.133;
   1:  PR[91,2] = PR[90,2] + -3.426;
   1:  PR[91,3] = PR[90,3] + 36.926;
   1:L PR[91] R[100]mm/sec CNT100;
   1:  PR[91,1] = PR[90,1] + -29.905;
   1:  PR[91,2] = PR[90,2] + -4.337;
   1:  PR[91,3] = PR[90,3] + 36.934;
   1:L PR[91] R[100]mm/sec CNT100;
   1:  PR[91,1] = PR[90,1] + -29.626;
   1:  PR[91,2] = PR[90,2] + -5.241;
   1:  PR[91,3] = PR[90,3] + 36.941;
   1:L PR[91] R[100]mm/sec CNT100;
   1:  PR[91,1] = PR[90,1] + -29.296;
   1:  PR[91,2] = PR[90,2] + -6.138;
   1:  PR[91,3] = PR[90,3] + 36.949;
   1:L PR[91] R[100]mm/sec CNT100;
   1:  PR[91,1] = PR[90,1] + -28.918;
   1:  PR[91,2] = PR[90,2] + -7.029;
   1:  PR[91,3] = PR[90,3] + 36.957;
   1:L PR[91] R[100]mm/sec CNT100;
   1:  PR[91,1] = PR[90,1] + -28.491;
   1:  PR[91,2] = PR[90,2] + -7.909;
   1:  PR[91,3] = PR[90,3] + 36.964;
   1:L PR[91] R[100]mm/sec CNT100;
   1:  PR[91,1] = PR[90,1] + -28.017;
   1:  PR[91,2] = PR[90,2] + -8.773;
   1:  PR[91,3] = PR[90,3] + 36.972;
   1:L PR[91] R[100]mm/sec CNT100;
   1:  PR[91,1] = PR[90,1] + -27.491;
   1:  PR[91,2] = PR[90,2] + -9.624;
   1:  PR[91,3] = PR[90,3] + 36.980;
   1:L PR[91] R[100]mm/sec CNT100;
   1:  PR[91,1] = PR[90,1] + -26.936;
   1:  PR[91,2] = PR[90,2] + -10.428;
   1:  PR[91,3] = PR[90,3] + 36.988;
   1:L PR[91] R[100]mm/sec CNT100;
   1:  PR[91,1] = PR[90,1] + -26.336;
   1:  PR[91,2] = PR[90,2] + -11.208;
   1:  PR[91,3] = PR[90,3] + 36.996;
   1:L PR[91] R[100]mm/sec CNT100;
   1:  PR[91,1] = PR[90,1] + -25.694;
   1:  PR[91,2] = PR[90,2] + -11.956;
   1:  PR[91,3] = PR[90,3] + 37.004;
   1:L PR[91] R[100]mm/sec CNT100;
   1:  PR[91,1] = PR[90,1] + -25.015;
   1:  PR[91,2] = PR[90,2] + -12.670;
   1:  PR[91,3] = PR[90,3] + 37.012;
   1:L PR[91] R[100]mm/sec CNT100;
   1:  PR[91,1] = PR[90,1] + -24.298;
   1:  PR[91,2] = PR[90,2] + -13.351;
   1:  PR[91,3] = PR[90,3] + 37.020;
   1:L PR[91] R[100]mm/sec CNT100;
   1:  PR[91,1] = PR[90,1] + -23.546;
   1:  PR[91,2] = PR[90,2] + -13.996;
   1:  PR[91,3] = PR[90,3] + 37.028;
   1:L PR[91] R[100]mm/sec CNT100;
   1:  PR[91,1] = PR[90,1] + -22.761;
   1:  PR[91,2] = PR[90,2] + -14.605;
   1:  PR[91,3] = PR[90,3] + 37.036;
   1:L PR[91] R[100]mm/sec CNT100;
   1:  PR[91,1] = PR[90,1] + -21.945;
   1:  PR[91,2] = PR[90,2] + -15.175;
   1:  PR[91,3] = PR[90,3] + 37.044;
   1:L PR[91] R[100]mm/sec CNT100;
   1:  PR[91,1] = PR[90,1] + -21.098;
   1:  PR[91,2] = PR[90,2] + -15.707;
   1:  PR[91,3] = PR[90,3] + 37.052;
   1:L PR[91] R[100]mm/sec CNT100;
   1:  PR[91,1] = PR[90,1] + -20.686;
   1:  PR[91,2] = PR[90,2] + -15.942;
   1:  PR[91,3] = PR[90,3] + 37.060;
   1:L PR[91] R[100]mm/sec CNT100;
   1:  PR[91,1] = PR[90,1] + -20.229;
   1:  PR[91,2] = PR[90,2] + -16.196;
   1:  PR[91,3] = PR[90,3] + 37.063;
   1:L PR[91] R[100]mm/sec CNT100;
   1:  PR[91,1] = PR[90,1] + -19.331;
   1:  PR[91,2] = PR[90,2] + -16.646;
   1:  PR[91,3] = PR[90,3] + 37.068;
   1:L PR[91] R[100]mm/sec CNT100;
   1:  PR[91,1] = PR[90,1] + -18.413;
   1:  PR[91,2] = PR[90,2] + -17.051;
   1:  PR[91,3] = PR[90,3] + 37.076;
   1:L PR[91] R[100]mm/sec CNT100;
   1:  PR[91,1] = PR[90,1] + -17.475;
   1:  PR[91,2] = PR[90,2] + -17.412;
   1:  PR[91,3] = PR[90,3] + 37.084;
   1:L PR[91] R[100]mm/sec CNT100;
   1:  PR[91,1] = PR[90,1] + -16.519;
   1:  PR[91,2] = PR[90,2] + -17.727;
   1:  PR[91,3] = PR[90,3] + 37.092;
   1:L PR[91] R[100]mm/sec CNT100;
   1:  PR[91,1] = PR[90,1] + -15.549;
   1:  PR[91,2] = PR[90,2] + -17.995;
   1:  PR[91,3] = PR[90,3] + 37.100;
   1:L PR[91] R[100]mm/sec CNT100;
   1:  PR[91,1] = PR[90,1] + -14.566;
   1:  PR[91,2] = PR[90,2] + -18.217;
   1:  PR[91,3] = PR[90,3] + 37.108;
   1:L PR[91] R[100]mm/sec CNT100;
   1:  PR[91,1] = PR[90,1] + -13.572;
   1:  PR[91,2] = PR[90,2] + -18.391;
   1:  PR[91,3] = PR[90,3] + 37.116;
   1:L PR[91] R[100]mm/sec CNT100;
   1:  PR[91,1] = PR[90,1] + -12.568;
   1:  PR[91,2] = PR[90,2] + -18.518;
   1:  PR[91,3] = PR[90,3] + 37.124;
   1:L PR[91] R[100]mm/sec CNT100;
   1:  PR[91,1] = PR[90,1] + -11.561;
   1:  PR[91,2] = PR[90,2] + -18.597;
   1:  PR[91,3] = PR[90,3] + 37.132;
   1:L PR[91] R[100]mm/sec CNT100;
   1:  PR[91,1] = PR[90,1] + -10.550;
   1:  PR[91,2] = PR[90,2] + -18.628;
   1:  PR[91,3] = PR[90,3] + 37.140;
   1:L PR[91] R[100]mm/sec CNT100;
   1:  PR[91,1] = PR[90,1] + -9.538;
   1:  PR[91,2] = PR[90,2] + -18.610;
   1:  PR[91,3] = PR[90,3] + 37.148;
   1:L PR[91] R[100]mm/sec CNT100;
   1:  PR[91,1] = PR[90,1] + -8.528;
   1:  PR[91,2] = PR[90,2] + -18.543;
   1:  PR[91,3] = PR[90,3] + 37.157;
   1:L PR[91] R[100]mm/sec CNT100;
   1:  PR[91,1] = PR[90,1] + -7.523;
   1:  PR[91,2] = PR[90,2] + -18.427;
   1:  PR[91,3] = PR[90,3] + 37.165;
   1:L PR[91] R[100]mm/sec CNT100;
   1:  PR[91,1] = PR[90,1] + -6.526;
   1:  PR[91,2] = PR[90,2] + -18.262;
   1:  PR[91,3] = PR[90,3] + 37.173;
   1:L PR[91] R[100]mm/sec CNT100;
   1:  PR[91,1] = PR[90,1] + -5.536;
   1:  PR[91,2] = PR[90,2] + -18.048;
   1:  PR[91,3] = PR[90,3] + 37.181;
   1:L PR[91] R[100]mm/sec CNT100;
   1:  PR[91,1] = PR[90,1] + -5.105;
   1:  PR[91,2] = PR[90,2] + -17.936;
   1:  PR[91,3] = PR[90,3] + 37.189;
   1:L PR[91] R[100]mm/sec CNT100;
   1:  PR[91,1] = PR[90,1] + -4.564;
   1:  PR[91,2] = PR[90,2] + -17.787;
   1:  PR[91,3] = PR[90,3] + 37.193;
   1:L PR[91] R[100]mm/sec CNT100;
   1:  PR[91,1] = PR[90,1] + -4.081;
   1:  PR[91,2] = PR[90,2] + -17.635;
   1:  PR[91,3] = PR[90,3] + 37.197;
   1:L PR[91] R[100]mm/sec CNT100;
   1:  PR[91,1] = PR[90,1] + -3.604;
   1:  PR[91,2] = PR[90,2] + -17.478;
   1:  PR[91,3] = PR[90,3] + 37.201;
   1:L PR[91] R[100]mm/sec CNT100;
   1:  PR[91,1] = PR[90,1] + -3.076;
   1:  PR[91,2] = PR[90,2] + -17.282;
   1:  PR[91,3] = PR[90,3] + 37.205;
   1:L PR[91] R[100]mm/sec CNT100;
   1:  PR[91,1] = PR[90,1] + -2.663;
   1:  PR[91,2] = PR[90,2] + -17.123;
   1:  PR[91,3] = PR[90,3] + 37.210;
   1:L PR[91] R[100]mm/sec CNT100;
   1:  PR[91,1] = PR[90,1] + -1.739;
   1:  PR[91,2] = PR[90,2] + -16.721;
   1:  PR[91,3] = PR[90,3] + 37.213;
   1:L PR[91] R[100]mm/sec CNT100;
   1:  PR[91,1] = PR[90,1] + -1.406;
   1:  PR[91,2] = PR[90,2] + -16.558;
   1:  PR[91,3] = PR[90,3] + 37.221;
   1:L PR[91] R[100]mm/sec CNT100;
   1:  PR[91,1] = PR[90,1] + -0.972;
   1:  PR[91,2] = PR[90,2] + -16.388;
   1:  PR[91,3] = PR[90,3] + 37.224;
   1:L PR[91] R[100]mm/sec CNT100;
   1:  PR[91,1] = PR[90,1] + -0.493;
   1:  PR[91,2] = PR[90,2] + -16.287;
   1:  PR[91,3] = PR[90,3] + 37.228;
   1:L PR[91] R[100]mm/sec CNT100;
   1:  PR[91,1] = PR[90,1] + -0.002;
   1:  PR[91,2] = PR[90,2] + -16.266;
   1:  PR[91,3] = PR[90,3] + 37.232;
   1:L PR[91] R[100]mm/sec CNT100;
   1:  PR[91,1] = PR[90,1] + 0.487;
   1:  PR[91,2] = PR[90,2] + -16.327;
   1:  PR[91,3] = PR[90,3] + 37.236;
   1:L PR[91] R[100]mm/sec CNT100;
   1:  PR[91] = PR[90];
   1:  PR[91,1] = PR[90,1] + 1.013;
   1:  PR[91,2] = PR[90,2] + -16.933;
   1:  PR[91,3] = PR[90,3] + 38.570;
   1:L PR[91] R[100]mm/sec CNT100;
   1:  PR[91,1] = PR[90,1] + 1.971;
   1:  PR[91,2] = PR[90,2] + -17.343;
   1:  PR[91,3] = PR[90,3] + 37.244;
   1:L PR[91] R[100]mm/sec CNT100;
   1:  PR[91,1] = PR[90,1] + 2.941;
   1:  PR[91,2] = PR[90,2] + -17.700;
   1:  PR[91,3] = PR[90,3] + 37.252;
   1:L PR[91] R[100]mm/sec CNT100;
   1:  PR[91,1] = PR[90,1] + 3.889;
   1:  PR[91,2] = PR[90,2] + -17.999;
   1:  PR[91,3] = PR[90,3] + 37.261;
   1:L PR[91] R[100]mm/sec CNT100;
   1:  PR[91,1] = PR[90,1] + 4.868;
   1:  PR[91,2] = PR[90,2] + -18.256;
   1:  PR[91,3] = PR[90,3] + 37.269;
   1:L PR[91] R[100]mm/sec CNT100;
   1:  PR[91,1] = PR[90,1] + 6.053;
   1:  PR[91,2] = PR[90,2] + -18.498;
   1:  PR[91,3] = PR[90,3] + 37.277;
   1:L PR[91] R[100]mm/sec CNT100;
   1:  PR[91,1] = PR[90,1] + 6.865;
   1:  PR[91,2] = PR[90,2] + -18.627;
   1:  PR[91,3] = PR[90,3] + 37.287;
   1:L PR[91] R[100]mm/sec CNT100;
   1:  PR[91,1] = PR[90,1] + 7.875;
   1:  PR[91,2] = PR[90,2] + -18.739;
   1:  PR[91,3] = PR[90,3] + 37.293;
   1:L PR[91] R[100]mm/sec CNT100;
   1:  PR[91,1] = PR[90,1] + 8.889;
   1:  PR[91,2] = PR[90,2] + -18.801;
   1:  PR[91,3] = PR[90,3] + 37.301;
   1:L PR[91] R[100]mm/sec CNT100;
   1:  PR[91,1] = PR[90,1] + 9.908;
   1:  PR[91,2] = PR[90,2] + -18.814;
   1:  PR[91,3] = PR[90,3] + 37.310;
   1:L PR[91] R[100]mm/sec CNT100;
   1:  PR[91,1] = PR[90,1] + 10.339;
   1:  PR[91,2] = PR[90,2] + -18.801;
   1:  PR[91,3] = PR[90,3] + 37.318;
   1:L PR[91] R[100]mm/sec CNT100;
   1:  PR[91,1] = PR[90,1] + 10.921;
   1:  PR[91,2] = PR[90,2] + -18.778;
   1:  PR[91,3] = PR[90,3] + 37.321;
   1:L PR[91] R[100]mm/sec CNT100;
   1:  PR[91,1] = PR[90,1] + 11.935;
   1:  PR[91,2] = PR[90,2] + -18.693;
   1:  PR[91,3] = PR[90,3] + 37.326;
   1:L PR[91] R[100]mm/sec CNT100;
   1:  PR[91,1] = PR[90,1] + 12.942;
   1:  PR[91,2] = PR[90,2] + -18.559;
   1:  PR[91,3] = PR[90,3] + 37.334;
   1:L PR[91] R[100]mm/sec CNT100;
   1:  PR[91,1] = PR[90,1] + 13.941;
   1:  PR[91,2] = PR[90,2] + -18.376;
   1:  PR[91,3] = PR[90,3] + 37.343;
   1:L PR[91] R[100]mm/sec CNT100;
   1:  PR[91,1] = PR[90,1] + 14.929;
   1:  PR[91,2] = PR[90,2] + -18.146;
   1:  PR[91,3] = PR[90,3] + 37.351;
   1:L PR[91] R[100]mm/sec CNT100;
   1:  PR[91,1] = PR[90,1] + 15.904;
   1:  PR[91,2] = PR[90,2] + -17.868;
   1:  PR[91,3] = PR[90,3] + 37.359;
   1:L PR[91] R[100]mm/sec CNT100;
   1:  PR[91,1] = PR[90,1] + 16.863;
   1:  PR[91,2] = PR[90,2] + -17.544;
   1:  PR[91,3] = PR[90,3] + 37.367;
   1:L PR[91] R[100]mm/sec CNT100;
   1:  PR[91,1] = PR[90,1] + 17.805;
   1:  PR[91,2] = PR[90,2] + -17.175;
   1:  PR[91,3] = PR[90,3] + 37.375;
   1:L PR[91] R[100]mm/sec CNT100;
   1:  PR[91,1] = PR[90,1] + 18.726;
   1:  PR[91,2] = PR[90,2] + -16.762;
   1:  PR[91,3] = PR[90,3] + 37.384;
   1:L PR[91] R[100]mm/sec CNT100;
   1:  PR[91,1] = PR[90,1] + 19.624;
   1:  PR[91,2] = PR[90,2] + -16.305;
   1:  PR[91,3] = PR[90,3] + 37.392;
   1:L PR[91] R[100]mm/sec CNT100;
   1:  PR[91,1] = PR[90,1] + 20.497;
   1:  PR[91,2] = PR[90,2] + -15.809;
   1:  PR[91,3] = PR[90,3] + 37.400;
   1:L PR[91] R[100]mm/sec CNT100;
   1:  PR[91,1] = PR[90,1] + 21.341;
   1:  PR[91,2] = PR[90,2] + -15.272;
   1:  PR[91,3] = PR[90,3] + 37.408;
   1:L PR[91] R[100]mm/sec CNT100;
   1:  PR[91,1] = PR[90,1] + 22.157;
   1:  PR[91,2] = PR[90,2] + -14.696;
   1:  PR[91,3] = PR[90,3] + 37.416;
   1:L PR[91] R[100]mm/sec CNT100;
   1:  PR[91,1] = PR[90,1] + 22.942;
   1:  PR[91,2] = PR[90,2] + -14.082;
   1:  PR[91,3] = PR[90,3] + 37.424;
   1:L PR[91] R[100]mm/sec CNT100;
   1:  PR[91,1] = PR[90,1] + 23.693;
   1:  PR[91,2] = PR[90,2] + -13.430;
   1:  PR[91,3] = PR[90,3] + 37.432;
   1:L PR[91] R[100]mm/sec CNT100;
   1:  PR[91,1] = PR[90,1] + 24.409;
   1:  PR[91,2] = PR[90,2] + -12.742;
   1:  PR[91,3] = PR[90,3] + 37.440;
   1:L PR[91] R[100]mm/sec CNT100;
   1:  PR[91,1] = PR[90,1] + 25.089;
   1:  PR[91,2] = PR[90,2] + -12.019;
   1:  PR[91,3] = PR[90,3] + 37.448;
   1:L PR[91] R[100]mm/sec CNT100;
   1:  PR[91,1] = PR[90,1] + 25.330;
   1:  PR[91,2] = PR[90,2] + -11.737;
   1:  PR[91,3] = PR[90,3] + 37.456;
   1:L PR[91] R[100]mm/sec CNT100;
   1:  PR[91,1] = PR[90,1] + 25.728;
   1:  PR[91,2] = PR[90,2] + -11.265;
   1:  PR[91,3] = PR[90,3] + 37.459;
   1:L PR[91] R[100]mm/sec CNT100;
   1:  PR[91,1] = PR[90,1] + 26.328;
   1:  PR[91,2] = PR[90,2] + -10.477;
   1:  PR[91,3] = PR[90,3] + 37.464;
   1:L PR[91] R[100]mm/sec CNT100;
   1:  PR[91,1] = PR[90,1] + 26.887;
   1:  PR[91,2] = PR[90,2] + -9.661;
   1:  PR[91,3] = PR[90,3] + 37.472;
   1:L PR[91] R[100]mm/sec CNT100;
   1:  PR[91,1] = PR[90,1] + 27.402;
   1:  PR[91,2] = PR[90,2] + -8.821;
   1:  PR[91,3] = PR[90,3] + 37.480;
   1:L PR[91] R[100]mm/sec CNT100;
   1:  PR[91,1] = PR[90,1] + 27.873;
   1:  PR[91,2] = PR[90,2] + -7.960;
   1:  PR[91,3] = PR[90,3] + 37.488;
   1:L PR[91] R[100]mm/sec CNT100;
   1:  PR[91,1] = PR[90,1] + 28.297;
   1:  PR[91,2] = PR[90,2] + -7.083;
   1:  PR[91,3] = PR[90,3] + 37.496;
   1:L PR[91] R[100]mm/sec CNT100;
   1:  PR[91,1] = PR[90,1] + 28.674;
   1:  PR[91,2] = PR[90,2] + -6.196;
   1:  PR[91,3] = PR[90,3] + 37.504;
   1:L PR[91] R[100]mm/sec CNT100;
   1:  PR[91,1] = PR[90,1] + 29.003;
   1:  PR[91,2] = PR[90,2] + -5.298;
   1:  PR[91,3] = PR[90,3] + 37.512;
   1:L PR[91] R[100]mm/sec CNT100;
   1:  PR[91,1] = PR[90,1] + 29.282;
   1:  PR[91,2] = PR[90,2] + -4.391;
   1:  PR[91,3] = PR[90,3] + 37.520;
   1:L PR[91] R[100]mm/sec CNT100;
   1:  PR[91,1] = PR[90,1] + 29.511;
   1:  PR[91,2] = PR[90,2] + -3.471;
   1:  PR[91,3] = PR[90,3] + 37.527;
   1:L PR[91] R[100]mm/sec CNT100;
   1:  PR[91,1] = PR[90,1] + 29.690;
   1:  PR[91,2] = PR[90,2] + -2.534;
   1:  PR[91,3] = PR[90,3] + 37.535;
   1:L PR[91] R[100]mm/sec CNT100;
   1:  PR[91,1] = PR[90,1] + 29.818;
   1:  PR[91,2] = PR[90,2] + -1.575;
   1:  PR[91,3] = PR[90,3] + 37.543;
   1:L PR[91] R[100]mm/sec CNT100;
   1:  PR[91,1] = PR[90,1] + 29.895;
   1:  PR[91,2] = PR[90,2] + -0.589;
   1:  PR[91,3] = PR[90,3] + 37.551;
   1:L PR[91] R[100]mm/sec CNT100;
   1:  PR[91,1] = PR[90,1] + 29.921;
   1:  PR[91,2] = PR[90,2] + 0.428;
   1:  PR[91,3] = PR[90,3] + 37.559;
   1:L PR[91] R[100]mm/sec CNT100;
   1:  PR[91,1] = PR[90,1] + 29.895;
   1:  PR[91,2] = PR[90,2] + 1.444;
   1:  PR[91,3] = PR[90,3] + 37.567;
   1:L PR[91] R[100]mm/sec CNT100;
   1:  PR[91,1] = PR[90,1] + 29.818;
   1:  PR[91,2] = PR[90,2] + 2.430;
   1:  PR[91,3] = PR[90,3] + 37.575;
   1:L PR[91] R[100]mm/sec CNT100;
   1:  PR[91,1] = PR[90,1] + 29.690;
   1:  PR[91,2] = PR[90,2] + 3.389;
   1:  PR[91,3] = PR[90,3] + 37.583;
   1:L PR[91] R[100]mm/sec CNT100;
   1:  PR[91,1] = PR[90,1] + 29.511;
   1:  PR[91,2] = PR[90,2] + 4.326;
   1:  PR[91,3] = PR[90,3] + 37.591;
   1:L PR[91] R[100]mm/sec CNT100;
   1:  PR[91,1] = PR[90,1] + 29.282;
   1:  PR[91,2] = PR[90,2] + 5.246;
   1:  PR[91,3] = PR[90,3] + 37.599;
   1:L PR[91] R[100]mm/sec CNT100;
   1:  PR[91,1] = PR[90,1] + 29.003;
   1:  PR[91,2] = PR[90,2] + 6.154;
   1:  PR[91,3] = PR[90,3] + 37.606;
   1:L PR[91] R[100]mm/sec CNT100;
   1:  PR[91,1] = PR[90,1] + 28.674;
   1:  PR[91,2] = PR[90,2] + 7.052;
   1:  PR[91,3] = PR[90,3] + 37.614;
   1:L PR[91] R[100]mm/sec CNT100;
   1:  PR[91,1] = PR[90,1] + 28.528;
   1:  PR[91,2] = PR[90,2] + 7.398;
   1:  PR[91,3] = PR[90,3] + 37.622;
   1:L PR[91] R[100]mm/sec CNT100;
   1:  PR[91,1] = PR[90,1] + 28.298;
   1:  PR[91,2] = PR[90,2] + 7.938;
   1:  PR[91,3] = PR[90,3] + 37.625;
   1:L PR[91] R[100]mm/sec CNT100;
   1:  PR[91,1] = PR[90,1] + 27.873;
   1:  PR[91,2] = PR[90,2] + 8.815;
   1:  PR[91,3] = PR[90,3] + 37.630;
   1:L PR[91] R[100]mm/sec CNT100;
   1:  PR[91,1] = PR[90,1] + 27.402;
   1:  PR[91,2] = PR[90,2] + 9.676;
   1:  PR[91,3] = PR[90,3] + 37.637;
   1:L PR[91] R[100]mm/sec CNT100;
   1:  PR[91,1] = PR[90,1] + 26.886;
   1:  PR[91,2] = PR[90,2] + 10.517;
   1:  PR[91,3] = PR[90,3] + 37.645;
   1:L PR[91] R[100]mm/sec CNT100;
   1:  PR[91,1] = PR[90,1] + 26.590;
   1:  PR[91,2] = PR[90,2] + 10.953;
   1:  PR[91,3] = PR[90,3] + 37.653;
   1:L PR[91] R[100]mm/sec CNT100;
   1:  PR[91,1] = PR[90,1] + 26.329;
   1:  PR[91,2] = PR[90,2] + 11.331;
   1:  PR[91,3] = PR[90,3] + 37.658;
   1:L PR[91] R[100]mm/sec CNT100;
   1:  PR[91,1] = PR[90,1] + 25.728;
   1:  PR[91,2] = PR[90,2] + 12.119;
   1:  PR[91,3] = PR[90,3] + 37.661;
   1:L PR[91] R[100]mm/sec CNT100;
   1:  PR[91,1] = PR[90,1] + 25.088;
   1:  PR[91,2] = PR[90,2] + 12.875;
   1:  PR[91,3] = PR[90,3] + 37.669;
   1:L PR[91] R[100]mm/sec CNT100;
   1:  PR[91,1] = PR[90,1] + 24.408;
   1:  PR[91,2] = PR[90,2] + 13.599;
   1:  PR[91,3] = PR[90,3] + 37.677;
   1:L PR[91] R[100]mm/sec CNT100;
   1:  PR[91,1] = PR[90,1] + 23.897;
   1:  PR[91,2] = PR[90,2] + 14.092;
   1:  PR[91,3] = PR[90,3] + 37.685;
   1:L PR[91] R[100]mm/sec CNT100;
   1:  PR[91,1] = PR[90,1] + 22.939;
   1:  PR[91,2] = PR[90,2] + 14.939;
   1:  PR[91,3] = PR[90,3] + 37.691;
   1:L PR[91] R[100]mm/sec CNT100;
   1:  PR[91,1] = PR[90,1] + 22.156;
   1:  PR[91,2] = PR[90,2] + 15.552;
   1:  PR[91,3] = PR[90,3] + 37.702;
   1:L PR[91] R[100]mm/sec CNT100;
   1:  PR[91,1] = PR[90,1] + 21.340;
   1:  PR[91,2] = PR[90,2] + 16.128;
   1:  PR[91,3] = PR[90,3] + 37.710;
   1:L PR[91] R[100]mm/sec CNT100;
   1:  PR[91,1] = PR[90,1] + 20.495;
   1:  PR[91,2] = PR[90,2] + 16.665;
   1:  PR[91,3] = PR[90,3] + 37.718;
   1:L PR[91] R[100]mm/sec CNT100;
   1:  PR[91,1] = PR[90,1] + 19.619;
   1:  PR[91,2] = PR[90,2] + 17.163;
   1:  PR[91,3] = PR[90,3] + 37.726;
   1:L PR[91] R[100]mm/sec CNT100;
   1:  PR[91,1] = PR[90,1] + 18.724;
   1:  PR[91,2] = PR[90,2] + 17.617;
   1:  PR[91,3] = PR[90,3] + 37.734;
   1:L PR[91] R[100]mm/sec CNT100;
   1:  PR[91,1] = PR[90,1] + 17.803;
   1:  PR[91,2] = PR[90,2] + 18.031;
   1:  PR[91,3] = PR[90,3] + 37.742;
   1:L PR[91] R[100]mm/sec CNT100;
   1:  PR[91,1] = PR[90,1] + 16.862;
   1:  PR[91,2] = PR[90,2] + 18.400;
   1:  PR[91,3] = PR[90,3] + 37.750;
   1:L PR[91] R[100]mm/sec CNT100;
   1:  PR[91,1] = PR[90,1] + 15.902;
   1:  PR[91,2] = PR[90,2] + 18.724;
   1:  PR[91,3] = PR[90,3] + 37.758;
   1:L PR[91] R[100]mm/sec CNT100;
   1:  PR[91,1] = PR[90,1] + 14.927;
   1:  PR[91,2] = PR[90,2] + 19.001;
   1:  PR[91,3] = PR[90,3] + 37.767;
   1:L PR[91] R[100]mm/sec CNT100;
   1:  PR[91,1] = PR[90,1] + 13.937;
   1:  PR[91,2] = PR[90,2] + 19.232;
   1:  PR[91,3] = PR[90,3] + 37.775;
   1:L PR[91] R[100]mm/sec CNT100;
   1:  PR[91,1] = PR[90,1] + 13.560;
   1:  PR[91,2] = PR[90,2] + 19.303;
   1:  PR[91,3] = PR[90,3] + 37.783;
   1:L PR[91] R[100]mm/sec CNT100;
   1:  PR[91,1] = PR[90,1] + 12.941;
   1:  PR[91,2] = PR[90,2] + 19.414;
   1:  PR[91,3] = PR[90,3] + 37.786;
   1:L PR[91] R[100]mm/sec CNT100;
   1:  PR[91,1] = PR[90,1] + 11.933;
   1:  PR[91,2] = PR[90,2] + 19.548;
   1:  PR[91,3] = PR[90,3] + 37.791;
   1:L PR[91] R[100]mm/sec CNT100;
   1:  PR[91,1] = PR[90,1] + 10.920;
   1:  PR[91,2] = PR[90,2] + 19.633;
   1:  PR[91,3] = PR[90,3] + 37.799;
   1:L PR[91] R[100]mm/sec CNT100;
   1:  PR[91,1] = PR[90,1] + 9.904;
   1:  PR[91,2] = PR[90,2] + 19.669;
   1:  PR[91,3] = PR[90,3] + 37.808;
   1:L PR[91] R[100]mm/sec CNT100;
   1:  PR[91,1] = PR[90,1] + 8.888;
   1:  PR[91,2] = PR[90,2] + 19.656;
   1:  PR[91,3] = PR[90,3] + 37.816;
   1:L PR[91] R[100]mm/sec CNT100;
   1:  PR[91,1] = PR[90,1] + 7.873;
   1:  PR[91,2] = PR[90,2] + 19.594;
   1:  PR[91,3] = PR[90,3] + 37.824;
   1:L PR[91] R[100]mm/sec CNT100;
   1:  PR[91,1] = PR[90,1] + 6.863;
   1:  PR[91,2] = PR[90,2] + 19.482;
   1:  PR[91,3] = PR[90,3] + 37.832;
   1:L PR[91] R[100]mm/sec CNT100;
   1:  PR[91,1] = PR[90,1] + 5.861;
   1:  PR[91,2] = PR[90,2] + 19.321;
   1:  PR[91,3] = PR[90,3] + 37.841;
   1:L PR[91] R[100]mm/sec CNT100;
   1:  PR[91,1] = PR[90,1] + 4.868;
   1:  PR[91,2] = PR[90,2] + 19.111;
   1:  PR[91,3] = PR[90,3] + 37.849;
   1:L PR[91] R[100]mm/sec CNT100;
   1:  PR[91,1] = PR[90,1] + 3.887;
   1:  PR[91,2] = PR[90,2] + 18.854;
   1:  PR[91,3] = PR[90,3] + 37.857;
   1:L PR[91] R[100]mm/sec CNT100;
   1:  PR[91,1] = PR[90,1] + 2.921;
   1:  PR[91,2] = PR[90,2] + 18.549;
   1:  PR[91,3] = PR[90,3] + 37.865;
   1:L PR[91] R[100]mm/sec CNT100;
   1:  PR[91,1] = PR[90,1] + 1.952;
   1:  PR[91,2] = PR[90,2] + 18.190;
   1:  PR[91,3] = PR[90,3] + 37.873;
   1:L PR[91] R[100]mm/sec CNT100;
   1:  PR[91,1] = PR[90,1] + 1.013;
   1:  PR[91,2] = PR[90,2] + 17.788;
   1:  PR[91,3] = PR[90,3] + 37.882;
   1:L PR[91] R[100]mm/sec CNT100;
   1:  PR[91,1] = PR[90,1] + 0.566;
   1:  PR[91,2] = PR[90,2] + 17.645;
   1:  PR[91,3] = PR[90,3] + 37.890;
   1:L PR[91] R[100]mm/sec CNT100;
   1:  PR[91,1] = PR[90,1] + 0.081;
   1:  PR[91,2] = PR[90,2] + 17.570;
   1:  PR[91,3] = PR[90,3] + 37.894;
   1:L PR[91] R[100]mm/sec CNT100;
   1:  PR[91,1] = PR[90,1] + -0.412;
   1:  PR[91,2] = PR[90,2] + 17.577;
   1:  PR[91,3] = PR[90,3] + 37.898;
   1:L PR[91] R[100]mm/sec CNT100;
   1:  PR[91,1] = PR[90,1] + -0.895;
   1:  PR[91,2] = PR[90,2] + 17.666;
   1:  PR[91,3] = PR[90,3] + 37.902;
   1:L PR[91] R[100]mm/sec CNT100;
   1:  PR[91,1] = PR[90,1] + -1.327;
   1:  PR[91,2] = PR[90,2] + 17.822;
   1:  PR[91,3] = PR[90,3] + 37.906;
   1:L PR[91] R[100]mm/sec CNT100;
   1:  PR[91,1] = PR[90,1] + -2.207;
   1:  PR[91,2] = PR[90,2] + 18.198;
   1:  PR[91,3] = PR[90,3] + 37.909;
   1:L PR[91] R[100]mm/sec CNT100;
   1:  PR[91,1] = PR[90,1] + -3.180;
   1:  PR[91,2] = PR[90,2] + 18.557;
   1:  PR[91,3] = PR[90,3] + 37.917;
   1:L PR[91] R[100]mm/sec CNT100;
   1:  PR[91,1] = PR[90,1] + -4.127;
   1:  PR[91,2] = PR[90,2] + 18.856;
   1:  PR[91,3] = PR[90,3] + 37.926;
   1:L PR[91] R[100]mm/sec CNT100;
   1:  PR[91,1] = PR[90,1] + -5.108;
   1:  PR[91,2] = PR[90,2] + 19.113;
   1:  PR[91,3] = PR[90,3] + 37.934;
   1:L PR[91] R[100]mm/sec CNT100;
   1:  PR[91,1] = PR[90,1] + -6.099;
   1:  PR[91,2] = PR[90,2] + 19.321;
   1:  PR[91,3] = PR[90,3] + 37.942;
   1:L PR[91] R[100]mm/sec CNT100;
   1:  PR[91,1] = PR[90,1] + -7.356;
   1:  PR[91,2] = PR[90,2] + 19.512;
   1:  PR[91,3] = PR[90,3] + 37.950;
   1:L PR[91] R[100]mm/sec CNT100;
   1:  PR[91,1] = PR[90,1] + -8.113;
   1:  PR[91,2] = PR[90,2] + 19.593;
   1:  PR[91,3] = PR[90,3] + 37.960;
   1:L PR[91] R[100]mm/sec CNT100;
   1:  PR[91,1] = PR[90,1] + -9.129;
   1:  PR[91,2] = PR[90,2] + 19.656;
   1:  PR[91,3] = PR[90,3] + 37.966;
   1:L PR[91] R[100]mm/sec CNT100;
   1:  PR[91,1] = PR[90,1] + -10.145;
   1:  PR[91,2] = PR[90,2] + 19.669;
   1:  PR[91,3] = PR[90,3] + 37.975;
   1:L PR[91] R[100]mm/sec CNT100;
   1:  PR[91,1] = PR[90,1] + -11.163;
   1:  PR[91,2] = PR[90,2] + 19.633;
   1:  PR[91,3] = PR[90,3] + 37.983;
   1:L PR[91] R[100]mm/sec CNT100;
   1:  PR[91,1] = PR[90,1] + -11.658;
   1:  PR[91,2] = PR[90,2] + 19.593;
   1:  PR[91,3] = PR[90,3] + 37.991;
   1:L PR[91] R[100]mm/sec CNT100;
   1:  PR[91,1] = PR[90,1] + -12.173;
   1:  PR[91,2] = PR[90,2] + 19.548;
   1:  PR[91,3] = PR[90,3] + 37.995;
   1:L PR[91] R[100]mm/sec CNT100;
   1:  PR[91,1] = PR[90,1] + -13.181;
   1:  PR[91,2] = PR[90,2] + 19.413;
   1:  PR[91,3] = PR[90,3] + 37.999;
   1:L PR[91] R[100]mm/sec CNT100;
   1:  PR[91,1] = PR[90,1] + -14.180;
   1:  PR[91,2] = PR[90,2] + 19.231;
   1:  PR[91,3] = PR[90,3] + 38.008;
   1:L PR[91] R[100]mm/sec CNT100;
   1:  PR[91,1] = PR[90,1] + -15.169;
   1:  PR[91,2] = PR[90,2] + 19.001;
   1:  PR[91,3] = PR[90,3] + 38.016;
   1:L PR[91] R[100]mm/sec CNT100;
   1:  PR[91,1] = PR[90,1] + -16.143;
   1:  PR[91,2] = PR[90,2] + 18.724;
   1:  PR[91,3] = PR[90,3] + 38.024;
   1:L PR[91] R[100]mm/sec CNT100;
   1:  PR[91,1] = PR[90,1] + -17.103;
   1:  PR[91,2] = PR[90,2] + 18.400;
   1:  PR[91,3] = PR[90,3] + 38.032;
   1:L PR[91] R[100]mm/sec CNT100;
   1:  PR[91,1] = PR[90,1] + -18.044;
   1:  PR[91,2] = PR[90,2] + 18.031;
   1:  PR[91,3] = PR[90,3] + 38.040;
   1:L PR[91] R[100]mm/sec CNT100;
   1:  PR[91,1] = PR[90,1] + -18.964;
   1:  PR[91,2] = PR[90,2] + 17.617;
   1:  PR[91,3] = PR[90,3] + 38.049;
   1:L PR[91] R[100]mm/sec CNT100;
   1:  PR[91,1] = PR[90,1] + -19.863;
   1:  PR[91,2] = PR[90,2] + 17.159;
   1:  PR[91,3] = PR[90,3] + 38.057;
   1:L PR[91] R[100]mm/sec CNT100;
   1:  PR[91,1] = PR[90,1] + -20.735;
   1:  PR[91,2] = PR[90,2] + 16.662;
   1:  PR[91,3] = PR[90,3] + 38.065;
   1:L PR[91] R[100]mm/sec CNT100;
   1:  PR[91,1] = PR[90,1] + -21.581;
   1:  PR[91,2] = PR[90,2] + 16.124;
   1:  PR[91,3] = PR[90,3] + 38.073;
   1:L PR[91] R[100]mm/sec CNT100;
   1:  PR[91,1] = PR[90,1] + -22.397;
   1:  PR[91,2] = PR[90,2] + 15.548;
   1:  PR[91,3] = PR[90,3] + 38.081;
   1:L PR[91] R[100]mm/sec CNT100;
   1:  PR[91,1] = PR[90,1] + -23.181;
   1:  PR[91,2] = PR[90,2] + 14.934;
   1:  PR[91,3] = PR[90,3] + 38.089;
   1:L PR[91] R[100]mm/sec CNT100;
   1:  PR[91,1] = PR[90,1] + -23.933;
   1:  PR[91,2] = PR[90,2] + 14.283;
   1:  PR[91,3] = PR[90,3] + 38.097;
   1:L PR[91] R[100]mm/sec CNT100;
   1:  PR[91,1] = PR[90,1] + -24.649;
   1:  PR[91,2] = PR[90,2] + 13.596;
   1:  PR[91,3] = PR[90,3] + 38.105;
   1:L PR[91] R[100]mm/sec CNT100;
   1:  PR[91,1] = PR[90,1] + -25.328;
   1:  PR[91,2] = PR[90,2] + 12.876;
   1:  PR[91,3] = PR[90,3] + 38.113;
   1:L PR[91] R[100]mm/sec CNT100;
   1:  PR[91,1] = PR[90,1] + -25.968;
   1:  PR[91,2] = PR[90,2] + 12.123;
   1:  PR[91,3] = PR[90,3] + 38.121;
   1:L PR[91] R[100]mm/sec CNT100;
   1:  PR[91,1] = PR[90,1] + -26.568;
   1:  PR[91,2] = PR[90,2] + 11.338;
   1:  PR[91,3] = PR[90,3] + 38.129;
   1:L PR[91] R[100]mm/sec CNT100;
   1:  PR[91,1] = PR[90,1] + -27.126;
   1:  PR[91,2] = PR[90,2] + 10.524;
   1:  PR[91,3] = PR[90,3] + 38.137;
   1:L PR[91] R[100]mm/sec CNT100;
   1:  PR[91,1] = PR[90,1] + -27.641;
   1:  PR[91,2] = PR[90,2] + 9.682;
   1:  PR[91,3] = PR[90,3] + 38.145;
   1:L PR[91] R[100]mm/sec CNT100;
   1:  PR[91,1] = PR[90,1] + -28.111;
   1:  PR[91,2] = PR[90,2] + 8.818;
   1:  PR[91,3] = PR[90,3] + 38.153;
   1:L PR[91] R[100]mm/sec CNT100;
   1:  PR[91,1] = PR[90,1] + -28.535;
   1:  PR[91,2] = PR[90,2] + 7.937;
   1:  PR[91,3] = PR[90,3] + 38.161;
   1:L PR[91] R[100]mm/sec CNT100;
   1:  PR[91,1] = PR[90,1] + -28.913;
   1:  PR[91,2] = PR[90,2] + 7.043;
   1:  PR[91,3] = PR[90,3] + 38.169;
   1:L PR[91] R[100]mm/sec CNT100;
   1:  PR[91,1] = PR[90,1] + -29.241;
   1:  PR[91,2] = PR[90,2] + 6.141;
   1:  PR[91,3] = PR[90,3] + 38.177;
   1:L PR[91] R[100]mm/sec CNT100;
   1:  PR[91,1] = PR[90,1] + -29.521;
   1:  PR[91,2] = PR[90,2] + 5.230;
   1:  PR[91,3] = PR[90,3] + 38.185;
   1:L PR[91] R[100]mm/sec CNT100;
   1:  PR[91,1] = PR[90,1] + -29.750;
   1:  PR[91,2] = PR[90,2] + 4.311;
   1:  PR[91,3] = PR[90,3] + 38.193;
   1:L PR[91] R[100]mm/sec CNT100;
   1:  PR[91,1] = PR[90,1] + -29.928;
   1:  PR[91,2] = PR[90,2] + 3.378;
   1:  PR[91,3] = PR[90,3] + 38.200;
   1:L PR[91] R[100]mm/sec CNT100;
   1:  PR[91,1] = PR[90,1] + -30.057;
   1:  PR[91,2] = PR[90,2] + 2.424;
   1:  PR[91,3] = PR[90,3] + 38.208;
   1:L PR[91] R[100]mm/sec CNT100;
   1:  PR[91,1] = PR[90,1] + -30.134;
   1:  PR[91,2] = PR[90,2] + 1.442;
   1:  PR[91,3] = PR[90,3] + 38.216;
   1:L PR[91] R[100]mm/sec CNT100;
   1:  PR[91,1] = PR[90,1] + -30.160;
   1:  PR[91,2] = PR[90,2] + 0.428;
   1:  PR[91,3] = PR[90,3] + 38.224;
   1:L PR[91] R[100]mm/sec CNT100;
   1:  PR[91,1] = PR[90,1] + -30.134;
   1:  PR[91,2] = PR[90,2] + -0.587;
   1:  PR[91,3] = PR[90,3] + 38.232;
   1:L PR[91] R[100]mm/sec CNT100;
   1:  PR[91,1] = PR[90,1] + -30.057;
   1:  PR[91,2] = PR[90,2] + -1.569;
   1:  PR[91,3] = PR[90,3] + 38.240;
   1:L PR[91] R[100]mm/sec CNT100;
   1:  PR[91,1] = PR[90,1] + -29.928;
   1:  PR[91,2] = PR[90,2] + -2.523;
   1:  PR[91,3] = PR[90,3] + 38.248;
   1:L PR[91] R[100]mm/sec CNT100;
   1:  PR[91,1] = PR[90,1] + -29.750;
   1:  PR[91,2] = PR[90,2] + -3.456;
   1:  PR[91,3] = PR[90,3] + 38.256;
   1:L PR[91] R[100]mm/sec CNT100;
   1:  PR[91,1] = PR[90,1] + -29.521;
   1:  PR[91,2] = PR[90,2] + -4.375;
   1:  PR[91,3] = PR[90,3] + 38.264;
   1:L PR[91] R[100]mm/sec CNT100;
   1:  PR[91,1] = PR[90,1] + -29.241;
   1:  PR[91,2] = PR[90,2] + -5.286;
   1:  PR[91,3] = PR[90,3] + 38.271;
   1:L PR[91] R[100]mm/sec CNT100;
   1:  PR[91,1] = PR[90,1] + -29.123;
   1:  PR[91,2] = PR[90,2] + -5.614;
   1:  PR[91,3] = PR[90,3] + 38.279;
   1:L PR[91] R[100]mm/sec CNT100;
   1:  PR[91,1] = PR[90,1] + -28.913;
   1:  PR[91,2] = PR[90,2] + -6.187;
   1:  PR[91,3] = PR[90,3] + 38.282;
   1:L PR[91] R[100]mm/sec CNT100;
   1:  PR[91,1] = PR[90,1] + -28.536;
   1:  PR[91,2] = PR[90,2] + -7.081;
   1:  PR[91,3] = PR[90,3] + 38.287;
   1:L PR[91] R[100]mm/sec CNT100;
   1:  PR[91,1] = PR[90,1] + -28.111;
   1:  PR[91,2] = PR[90,2] + -7.963;
   1:  PR[91,3] = PR[90,3] + 38.295;
   1:L PR[91] R[100]mm/sec CNT100;
   1:  PR[91,1] = PR[90,1] + -27.641;
   1:  PR[91,2] = PR[90,2] + -8.827;
   1:  PR[91,3] = PR[90,3] + 38.302;
   1:L PR[91] R[100]mm/sec CNT100;
   1:  PR[91,1] = PR[90,1] + -27.126;
   1:  PR[91,2] = PR[90,2] + -9.669;
   1:  PR[91,3] = PR[90,3] + 38.310;
   1:L PR[91] R[100]mm/sec CNT100;
   1:  PR[91,1] = PR[90,1] + -26.829;
   1:  PR[91,2] = PR[90,2] + -10.105;
   1:  PR[91,3] = PR[90,3] + 38.318;
   1:L PR[91] R[100]mm/sec CNT100;
   1:  PR[91,1] = PR[90,1] + -26.569;
   1:  PR[91,2] = PR[90,2] + -10.482;
   1:  PR[91,3] = PR[90,3] + 38.323;
   1:L PR[91] R[100]mm/sec CNT100;
   1:  PR[91,1] = PR[90,1] + -25.969;
   1:  PR[91,2] = PR[90,2] + -11.267;
   1:  PR[91,3] = PR[90,3] + 38.326;
   1:L PR[91] R[100]mm/sec CNT100;
   1:  PR[91,1] = PR[90,1] + -25.328;
   1:  PR[91,2] = PR[90,2] + -12.020;
   1:  PR[91,3] = PR[90,3] + 38.334;
   1:L PR[91] R[100]mm/sec CNT100;
   1:  PR[91,1] = PR[90,1] + -24.649;
   1:  PR[91,2] = PR[90,2] + -12.741;
   1:  PR[91,3] = PR[90,3] + 38.342;
   1:L PR[91] R[100]mm/sec CNT100;
   1:  PR[91,1] = PR[90,1] + -23.933;
   1:  PR[91,2] = PR[90,2] + -13.427;
   1:  PR[91,3] = PR[90,3] + 38.350;
   1:L PR[91] R[100]mm/sec CNT100;
   1:  PR[91,1] = PR[90,1] + -23.356;
   1:  PR[91,2] = PR[90,2] + -13.929;
   1:  PR[91,3] = PR[90,3] + 38.358;
   1:L PR[91] R[100]mm/sec CNT100;
   1:  PR[91,1] = PR[90,1] + -22.396;
   1:  PR[91,2] = PR[90,2] + -14.694;
   1:  PR[91,3] = PR[90,3] + 38.365;
   1:L PR[91] R[100]mm/sec CNT100;
   1:  PR[91,1] = PR[90,1] + -21.582;
   1:  PR[91,2] = PR[90,2] + -15.269;
   1:  PR[91,3] = PR[90,3] + 38.375;
   1:L PR[91] R[100]mm/sec CNT100;
   1:  PR[91,1] = PR[90,1] + -20.737;
   1:  PR[91,2] = PR[90,2] + -15.806;
   1:  PR[91,3] = PR[90,3] + 38.383;
   1:L PR[91] R[100]mm/sec CNT100;
   1:  PR[91,1] = PR[90,1] + -19.861;
   1:  PR[91,2] = PR[90,2] + -16.305;
   1:  PR[91,3] = PR[90,3] + 38.391;
   1:L PR[91] R[100]mm/sec CNT100;
   1:  PR[91,1] = PR[90,1] + -18.966;
   1:  PR[91,2] = PR[90,2] + -16.761;
   1:  PR[91,3] = PR[90,3] + 38.399;
   1:L PR[91] R[100]mm/sec CNT100;
   1:  PR[91,1] = PR[90,1] + -18.045;
   1:  PR[91,2] = PR[90,2] + -17.175;
   1:  PR[91,3] = PR[90,3] + 38.407;
   1:L PR[91] R[100]mm/sec CNT100;
   1:  PR[91,1] = PR[90,1] + -17.104;
   1:  PR[91,2] = PR[90,2] + -17.545;
   1:  PR[91,3] = PR[90,3] + 38.415;
   1:L PR[91] R[100]mm/sec CNT100;
   1:  PR[91,1] = PR[90,1] + -16.145;
   1:  PR[91,2] = PR[90,2] + -17.869;
   1:  PR[91,3] = PR[90,3] + 38.423;
   1:L PR[91] R[100]mm/sec CNT100;
   1:  PR[91,1] = PR[90,1] + -15.170;
   1:  PR[91,2] = PR[90,2] + -18.146;
   1:  PR[91,3] = PR[90,3] + 38.432;
   1:L PR[91] R[100]mm/sec CNT100;
   1:  PR[91,1] = PR[90,1] + -14.182;
   1:  PR[91,2] = PR[90,2] + -18.376;
   1:  PR[91,3] = PR[90,3] + 38.440;
   1:L PR[91] R[100]mm/sec CNT100;
   1:  PR[91,1] = PR[90,1] + -13.183;
   1:  PR[91,2] = PR[90,2] + -18.558;
   1:  PR[91,3] = PR[90,3] + 38.448;
   1:L PR[91] R[100]mm/sec CNT100;
   1:  PR[91,1] = PR[90,1] + -12.176;
   1:  PR[91,2] = PR[90,2] + -18.692;
   1:  PR[91,3] = PR[90,3] + 38.456;
   1:L PR[91] R[100]mm/sec CNT100;
   1:  PR[91,1] = PR[90,1] + -11.163;
   1:  PR[91,2] = PR[90,2] + -18.777;
   1:  PR[91,3] = PR[90,3] + 38.464;
   1:L PR[91] R[100]mm/sec CNT100;
   1:  PR[91,1] = PR[90,1] + -10.147;
   1:  PR[91,2] = PR[90,2] + -18.814;
   1:  PR[91,3] = PR[90,3] + 38.473;
   1:L PR[91] R[100]mm/sec CNT100;
   1:  PR[91,1] = PR[90,1] + -9.131;
   1:  PR[91,2] = PR[90,2] + -18.801;
   1:  PR[91,3] = PR[90,3] + 38.481;
   1:L PR[91] R[100]mm/sec CNT100;
   1:  PR[91,1] = PR[90,1] + -8.116;
   1:  PR[91,2] = PR[90,2] + -18.738;
   1:  PR[91,3] = PR[90,3] + 38.489;
   1:L PR[91] R[100]mm/sec CNT100;
   1:  PR[91,1] = PR[90,1] + -7.106;
   1:  PR[91,2] = PR[90,2] + -18.627;
   1:  PR[91,3] = PR[90,3] + 38.497;
   1:L PR[91] R[100]mm/sec CNT100;
   1:  PR[91,1] = PR[90,1] + -6.103;
   1:  PR[91,2] = PR[90,2] + -18.467;
   1:  PR[91,3] = PR[90,3] + 38.506;
   1:L PR[91] R[100]mm/sec CNT100;
   1:  PR[91,1] = PR[90,1] + -5.110;
   1:  PR[91,2] = PR[90,2] + -18.258;
   1:  PR[91,3] = PR[90,3] + 38.514;
   1:L PR[91] R[100]mm/sec CNT100;
   1:  PR[91,1] = PR[90,1] + -4.129;
   1:  PR[91,2] = PR[90,2] + -18.001;
   1:  PR[91,3] = PR[90,3] + 38.522;
   1:L PR[91] R[100]mm/sec CNT100;
   1:  PR[91,1] = PR[90,1] + -3.163;
   1:  PR[91,2] = PR[90,2] + -17.696;
   1:  PR[91,3] = PR[90,3] + 38.530;
   1:L PR[91] R[100]mm/sec CNT100;
   1:  PR[91,1] = PR[90,1] + -2.191;
   1:  PR[91,2] = PR[90,2] + -17.336;
   1:  PR[91,3] = PR[90,3] + 38.538;
   1:L PR[91] R[100]mm/sec CNT100;
   1:  PR[91,1] = PR[90,1] + -1.326;
   1:  PR[91,2] = PR[90,2] + -16.967;
   1:  PR[91,3] = PR[90,3] + 38.547;
   1:L PR[91] R[100]mm/sec CNT100;
   1:  PR[91,1] = PR[90,1] + -0.895;
   1:  PR[91,2] = PR[90,2] + -16.810;
   1:  PR[91,3] = PR[90,3] + 38.554;
   1:L PR[91] R[100]mm/sec CNT100;
   1:  PR[91,1] = PR[90,1] + -0.412;
   1:  PR[91,2] = PR[90,2] + -16.722;
   1:  PR[91,3] = PR[90,3] + 38.558;
   1:L PR[91] R[100]mm/sec CNT100;
   1:  PR[91,1] = PR[90,1] + 0.081;
   1:  PR[91,2] = PR[90,2] + -16.714;
   1:  PR[91,3] = PR[90,3] + 38.562;
   1:L PR[91] R[100]mm/sec CNT100;
   1:  PR[91,1] = PR[90,1] + 0.566;
   1:  PR[91,2] = PR[90,2] + -16.790;
   1:  PR[91,3] = PR[90,3] + 38.566;
   1:L PR[91] R[100]mm/sec CNT100;
   1:  PR[91] = PR[90];
   1:  PR[91,1] = PR[90,1] + 2.470;
   1:  PR[91,2] = PR[90,2] + -17.921;
   1:  PR[91,3] = PR[90,3] + 39.900;
   1:L PR[91] R[100]mm/sec CNT100;
   1:  PR[91,1] = PR[90,1] + 3.453;
   1:  PR[91,2] = PR[90,2] + -18.224;
   1:  PR[91,3] = PR[90,3] + 38.586;
   1:L PR[91] R[100]mm/sec CNT100;
   1:  PR[91,1] = PR[90,1] + 4.450;
   1:  PR[91,2] = PR[90,2] + -18.478;
   1:  PR[91,3] = PR[90,3] + 38.594;
   1:L PR[91] R[100]mm/sec CNT100;
   1:  PR[91,1] = PR[90,1] + 5.456;
   1:  PR[91,2] = PR[90,2] + -18.683;
   1:  PR[91,3] = PR[90,3] + 38.603;
   1:L PR[91] R[100]mm/sec CNT100;
   1:  PR[91,1] = PR[90,1] + 6.211;
   1:  PR[91,2] = PR[90,2] + -18.800;
   1:  PR[91,3] = PR[90,3] + 38.611;
   1:L PR[91] R[100]mm/sec CNT100;
   1:  PR[91,1] = PR[90,1] + 7.486;
   1:  PR[91,2] = PR[90,2] + -18.941;
   1:  PR[91,3] = PR[90,3] + 38.617;
   1:L PR[91] R[100]mm/sec CNT100;
   1:  PR[91,1] = PR[90,1] + 8.500;
   1:  PR[91,2] = PR[90,2] + -18.995;
   1:  PR[91,3] = PR[90,3] + 38.628;
   1:L PR[91] R[100]mm/sec CNT100;
   1:  PR[91,1] = PR[90,1] + 9.515;
   1:  PR[91,2] = PR[90,2] + -19.001;
   1:  PR[91,3] = PR[90,3] + 38.636;
   1:L PR[91] R[100]mm/sec CNT100;
   1:  PR[91,1] = PR[90,1] + 10.526;
   1:  PR[91,2] = PR[90,2] + -18.958;
   1:  PR[91,3] = PR[90,3] + 38.644;
   1:L PR[91] R[100]mm/sec CNT100;
   1:  PR[91,1] = PR[90,1] + 11.541;
   1:  PR[91,2] = PR[90,2] + -18.867;
   1:  PR[91,3] = PR[90,3] + 38.652;
   1:L PR[91] R[100]mm/sec CNT100;
   1:  PR[91,1] = PR[90,1] + 12.552;
   1:  PR[91,2] = PR[90,2] + -18.728;
   1:  PR[91,3] = PR[90,3] + 38.661;
   1:L PR[91] R[100]mm/sec CNT100;
   1:  PR[91,1] = PR[90,1] + 13.554;
   1:  PR[91,2] = PR[90,2] + -18.540;
   1:  PR[91,3] = PR[90,3] + 38.669;
   1:L PR[91] R[100]mm/sec CNT100;
   1:  PR[91,1] = PR[90,1] + 14.545;
   1:  PR[91,2] = PR[90,2] + -18.303;
   1:  PR[91,3] = PR[90,3] + 38.677;
   1:L PR[91] R[100]mm/sec CNT100;
   1:  PR[91,1] = PR[90,1] + 15.523;
   1:  PR[91,2] = PR[90,2] + -18.020;
   1:  PR[91,3] = PR[90,3] + 38.686;
   1:L PR[91] R[100]mm/sec CNT100;
   1:  PR[91,1] = PR[90,1] + 16.486;
   1:  PR[91,2] = PR[90,2] + -17.690;
   1:  PR[91,3] = PR[90,3] + 38.694;
   1:L PR[91] R[100]mm/sec CNT100;
   1:  PR[91,1] = PR[90,1] + 17.429;
   1:  PR[91,2] = PR[90,2] + -17.315;
   1:  PR[91,3] = PR[90,3] + 38.702;
   1:L PR[91] R[100]mm/sec CNT100;
   1:  PR[91,1] = PR[90,1] + 18.353;
   1:  PR[91,2] = PR[90,2] + -16.895;
   1:  PR[91,3] = PR[90,3] + 38.711;
   1:L PR[91] R[100]mm/sec CNT100;
   1:  PR[91,1] = PR[90,1] + 18.774;
   1:  PR[91,2] = PR[90,2] + -16.682;
   1:  PR[91,3] = PR[90,3] + 38.719;
   1:L PR[91] R[100]mm/sec CNT100;
   1:  PR[91,1] = PR[90,1] + 19.251;
   1:  PR[91,2] = PR[90,2] + -16.434;
   1:  PR[91,3] = PR[90,3] + 38.723;
   1:L PR[91] R[100]mm/sec CNT100;
   1:  PR[91,1] = PR[90,1] + 20.127;
   1:  PR[91,2] = PR[90,2] + -15.929;
   1:  PR[91,3] = PR[90,3] + 38.727;
   1:L PR[91] R[100]mm/sec CNT100;
   1:  PR[91,1] = PR[90,1] + 20.974;
   1:  PR[91,2] = PR[90,2] + -15.384;
   1:  PR[91,3] = PR[90,3] + 38.735;
   1:L PR[91] R[100]mm/sec CNT100;
   1:  PR[91,1] = PR[90,1] + 21.791;
   1:  PR[91,2] = PR[90,2] + -14.800;
   1:  PR[91,3] = PR[90,3] + 38.744;
   1:L PR[91] R[100]mm/sec CNT100;
   1:  PR[91,1] = PR[90,1] + 22.576;
   1:  PR[91,2] = PR[90,2] + -14.177;
   1:  PR[91,3] = PR[90,3] + 38.752;
   1:L PR[91] R[100]mm/sec CNT100;
   1:  PR[91,1] = PR[90,1] + 23.328;
   1:  PR[91,2] = PR[90,2] + -13.517;
   1:  PR[91,3] = PR[90,3] + 38.760;
   1:L PR[91] R[100]mm/sec CNT100;
   1:  PR[91,1] = PR[90,1] + 24.044;
   1:  PR[91,2] = PR[90,2] + -12.821;
   1:  PR[91,3] = PR[90,3] + 38.768;
   1:L PR[91] R[100]mm/sec CNT100;
   1:  PR[91,1] = PR[90,1] + 24.723;
   1:  PR[91,2] = PR[90,2] + -12.091;
   1:  PR[91,3] = PR[90,3] + 38.776;
   1:L PR[91] R[100]mm/sec CNT100;
   1:  PR[91,1] = PR[90,1] + 25.362;
   1:  PR[91,2] = PR[90,2] + -11.328;
   1:  PR[91,3] = PR[90,3] + 38.784;
   1:L PR[91] R[100]mm/sec CNT100;
   1:  PR[91,1] = PR[90,1] + 25.961;
   1:  PR[91,2] = PR[90,2] + -10.534;
   1:  PR[91,3] = PR[90,3] + 38.792;
   1:L PR[91] R[100]mm/sec CNT100;
   1:  PR[91,1] = PR[90,1] + 26.518;
   1:  PR[91,2] = PR[90,2] + -9.713;
   1:  PR[91,3] = PR[90,3] + 38.801;
   1:L PR[91] R[100]mm/sec CNT100;
   1:  PR[91,1] = PR[90,1] + 27.033;
   1:  PR[91,2] = PR[90,2] + -8.865;
   1:  PR[91,3] = PR[90,3] + 38.809;
   1:L PR[91] R[100]mm/sec CNT100;
   1:  PR[91,1] = PR[90,1] + 27.502;
   1:  PR[91,2] = PR[90,2] + -8.001;
   1:  PR[91,3] = PR[90,3] + 38.817;
   1:L PR[91] R[100]mm/sec CNT100;
   1:  PR[91,1] = PR[90,1] + 27.926;
   1:  PR[91,2] = PR[90,2] + -7.120;
   1:  PR[91,3] = PR[90,3] + 38.825;
   1:L PR[91] R[100]mm/sec CNT100;
   1:  PR[91,1] = PR[90,1] + 28.302;
   1:  PR[91,2] = PR[90,2] + -6.227;
   1:  PR[91,3] = PR[90,3] + 38.833;
   1:L PR[91] R[100]mm/sec CNT100;
   1:  PR[91,1] = PR[90,1] + 28.630;
   1:  PR[91,2] = PR[90,2] + -5.325;
   1:  PR[91,3] = PR[90,3] + 38.841;
   1:L PR[91] R[100]mm/sec CNT100;
   1:  PR[91,1] = PR[90,1] + 28.908;
   1:  PR[91,2] = PR[90,2] + -4.412;
   1:  PR[91,3] = PR[90,3] + 38.848;
   1:L PR[91] R[100]mm/sec CNT100;
   1:  PR[91,1] = PR[90,1] + 29.137;
   1:  PR[91,2] = PR[90,2] + -3.485;
   1:  PR[91,3] = PR[90,3] + 38.856;
   1:L PR[91] R[100]mm/sec CNT100;
   1:  PR[91,1] = PR[90,1] + 29.316;
   1:  PR[91,2] = PR[90,2] + -2.543;
   1:  PR[91,3] = PR[90,3] + 38.864;
   1:L PR[91] R[100]mm/sec CNT100;
   1:  PR[91,1] = PR[90,1] + 29.444;
   1:  PR[91,2] = PR[90,2] + -1.579;
   1:  PR[91,3] = PR[90,3] + 38.872;
   1:L PR[91] R[100]mm/sec CNT100;
   1:  PR[91,1] = PR[90,1] + 29.521;
   1:  PR[91,2] = PR[90,2] + -0.590;
   1:  PR[91,3] = PR[90,3] + 38.880;
   1:L PR[91] R[100]mm/sec CNT100;
   1:  PR[91,1] = PR[90,1] + 29.547;
   1:  PR[91,2] = PR[90,2] + 0.428;
   1:  PR[91,3] = PR[90,3] + 38.888;
   1:L PR[91] R[100]mm/sec CNT100;
   1:  PR[91,1] = PR[90,1] + 29.521;
   1:  PR[91,2] = PR[90,2] + 1.445;
   1:  PR[91,3] = PR[90,3] + 38.896;
   1:L PR[91] R[100]mm/sec CNT100;
   1:  PR[91,1] = PR[90,1] + 29.444;
   1:  PR[91,2] = PR[90,2] + 2.434;
   1:  PR[91,3] = PR[90,3] + 38.904;
   1:L PR[91] R[100]mm/sec CNT100;
   1:  PR[91,1] = PR[90,1] + 29.315;
   1:  PR[91,2] = PR[90,2] + 3.398;
   1:  PR[91,3] = PR[90,3] + 38.913;
   1:L PR[91] R[100]mm/sec CNT100;
   1:  PR[91,1] = PR[90,1] + 29.137;
   1:  PR[91,2] = PR[90,2] + 4.341;
   1:  PR[91,3] = PR[90,3] + 38.920;
   1:L PR[91] R[100]mm/sec CNT100;
   1:  PR[91,1] = PR[90,1] + 28.908;
   1:  PR[91,2] = PR[90,2] + 5.267;
   1:  PR[91,3] = PR[90,3] + 38.928;
   1:L PR[91] R[100]mm/sec CNT100;
   1:  PR[91,1] = PR[90,1] + 28.630;
   1:  PR[91,2] = PR[90,2] + 6.180;
   1:  PR[91,3] = PR[90,3] + 38.936;
   1:L PR[91] R[100]mm/sec CNT100;
   1:  PR[91,1] = PR[90,1] + 28.302;
   1:  PR[91,2] = PR[90,2] + 7.083;
   1:  PR[91,3] = PR[90,3] + 38.944;
   1:L PR[91] R[100]mm/sec CNT100;
   1:  PR[91,1] = PR[90,1] + 27.926;
   1:  PR[91,2] = PR[90,2] + 7.975;
   1:  PR[91,3] = PR[90,3] + 38.952;
   1:L PR[91] R[100]mm/sec CNT100;
   1:  PR[91,1] = PR[90,1] + 27.502;
   1:  PR[91,2] = PR[90,2] + 8.857;
   1:  PR[91,3] = PR[90,3] + 38.960;
   1:L PR[91] R[100]mm/sec CNT100;
   1:  PR[91,1] = PR[90,1] + 27.032;
   1:  PR[91,2] = PR[90,2] + 9.722;
   1:  PR[91,3] = PR[90,3] + 38.968;
   1:L PR[91] R[100]mm/sec CNT100;
   1:  PR[91,1] = PR[90,1] + 26.518;
   1:  PR[91,2] = PR[90,2] + 10.569;
   1:  PR[91,3] = PR[90,3] + 38.976;
   1:L PR[91] R[100]mm/sec CNT100;
   1:  PR[91,1] = PR[90,1] + 25.961;
   1:  PR[91,2] = PR[90,2] + 11.390;
   1:  PR[91,3] = PR[90,3] + 38.984;
   1:L PR[91] R[100]mm/sec CNT100;
   1:  PR[91,1] = PR[90,1] + 25.362;
   1:  PR[91,2] = PR[90,2] + 12.184;
   1:  PR[91,3] = PR[90,3] + 38.992;
   1:L PR[91] R[100]mm/sec CNT100;
   1:  PR[91,1] = PR[90,1] + 24.723;
   1:  PR[91,2] = PR[90,2] + 12.945;
   1:  PR[91,3] = PR[90,3] + 39.000;
   1:L PR[91] R[100]mm/sec CNT100;
   1:  PR[91,1] = PR[90,1] + 23.892;
   1:  PR[91,2] = PR[90,2] + 13.826;
   1:  PR[91,3] = PR[90,3] + 39.008;
   1:L PR[91] R[100]mm/sec CNT100;
   1:  PR[91,1] = PR[90,1] + 23.327;
   1:  PR[91,2] = PR[90,2] + 14.373;
   1:  PR[91,3] = PR[90,3] + 39.018;
   1:L PR[91] R[100]mm/sec CNT100;
   1:  PR[91,1] = PR[90,1] + 22.575;
   1:  PR[91,2] = PR[90,2] + 15.033;
   1:  PR[91,3] = PR[90,3] + 39.024;
   1:L PR[91] R[100]mm/sec CNT100;
   1:  PR[91,1] = PR[90,1] + 21.790;
   1:  PR[91,2] = PR[90,2] + 15.655;
   1:  PR[91,3] = PR[90,3] + 39.032;
   1:L PR[91] R[100]mm/sec CNT100;
   1:  PR[91,1] = PR[90,1] + 20.973;
   1:  PR[91,2] = PR[90,2] + 16.240;
   1:  PR[91,3] = PR[90,3] + 39.041;
   1:L PR[91] R[100]mm/sec CNT100;
   1:  PR[91,1] = PR[90,1] + 20.125;
   1:  PR[91,2] = PR[90,2] + 16.786;
   1:  PR[91,3] = PR[90,3] + 39.049;
   1:L PR[91] R[100]mm/sec CNT100;
   1:  PR[91,1] = PR[90,1] + 19.712;
   1:  PR[91,2] = PR[90,2] + 17.026;
   1:  PR[91,3] = PR[90,3] + 39.057;
   1:L PR[91] R[100]mm/sec CNT100;
   1:  PR[91,1] = PR[90,1] + 19.252;
   1:  PR[91,2] = PR[90,2] + 17.289;
   1:  PR[91,3] = PR[90,3] + 39.061;
   1:L PR[91] R[100]mm/sec CNT100;
   1:  PR[91,1] = PR[90,1] + 18.351;
   1:  PR[91,2] = PR[90,2] + 17.752;
   1:  PR[91,3] = PR[90,3] + 39.065;
   1:L PR[91] R[100]mm/sec CNT100;
   1:  PR[91,1] = PR[90,1] + 17.428;
   1:  PR[91,2] = PR[90,2] + 18.171;
   1:  PR[91,3] = PR[90,3] + 39.073;
   1:L PR[91] R[100]mm/sec CNT100;
   1:  PR[91,1] = PR[90,1] + 16.484;
   1:  PR[91,2] = PR[90,2] + 18.546;
   1:  PR[91,3] = PR[90,3] + 39.082;
   1:L PR[91] R[100]mm/sec CNT100;
   1:  PR[91,1] = PR[90,1] + 15.522;
   1:  PR[91,2] = PR[90,2] + 18.876;
   1:  PR[91,3] = PR[90,3] + 39.090;
   1:L PR[91] R[100]mm/sec CNT100;
   1:  PR[91,1] = PR[90,1] + 14.544;
   1:  PR[91,2] = PR[90,2] + 19.159;
   1:  PR[91,3] = PR[90,3] + 39.098;
   1:L PR[91] R[100]mm/sec CNT100;
   1:  PR[91,1] = PR[90,1] + 13.723;
   1:  PR[91,2] = PR[90,2] + 19.356;
   1:  PR[91,3] = PR[90,3] + 39.107;
   1:L PR[91] R[100]mm/sec CNT100;
   1:  PR[91,1] = PR[90,1] + 12.549;
   1:  PR[91,2] = PR[90,2] + 19.583;
   1:  PR[91,3] = PR[90,3] + 39.114;
   1:L PR[91] R[100]mm/sec CNT100;
   1:  PR[91,1] = PR[90,1] + 11.540;
   1:  PR[91,2] = PR[90,2] + 19.722;
   1:  PR[91,3] = PR[90,3] + 39.123;
   1:L PR[91] R[100]mm/sec CNT100;
   1:  PR[91,1] = PR[90,1] + 10.513;
   1:  PR[91,2] = PR[90,2] + 19.814;
   1:  PR[91,3] = PR[90,3] + 39.132;
   1:L PR[91] R[100]mm/sec CNT100;
   1:  PR[91,1] = PR[90,1] + 9.515;
   1:  PR[91,2] = PR[90,2] + 19.856;
   1:  PR[91,3] = PR[90,3] + 39.140;
   1:L PR[91] R[100]mm/sec CNT100;
   1:  PR[91,1] = PR[90,1] + 8.362;
   1:  PR[91,2] = PR[90,2] + 19.845;
   1:  PR[91,3] = PR[90,3] + 39.148;
   1:L PR[91] R[100]mm/sec CNT100;
   1:  PR[91,1] = PR[90,1] + 7.482;
   1:  PR[91,2] = PR[90,2] + 19.796;
   1:  PR[91,3] = PR[90,3] + 39.158;
   1:L PR[91] R[100]mm/sec CNT100;
   1:  PR[91,1] = PR[90,1] + 6.466;
   1:  PR[91,2] = PR[90,2] + 19.692;
   1:  PR[91,3] = PR[90,3] + 39.165;
   1:L PR[91] R[100]mm/sec CNT100;
   1:  PR[91,1] = PR[90,1] + 5.454;
   1:  PR[91,2] = PR[90,2] + 19.537;
   1:  PR[91,3] = PR[90,3] + 39.173;
   1:L PR[91] R[100]mm/sec CNT100;
   1:  PR[91,1] = PR[90,1] + 4.449;
   1:  PR[91,2] = PR[90,2] + 19.333;
   1:  PR[91,3] = PR[90,3] + 39.181;
   1:L PR[91] R[100]mm/sec CNT100;
   1:  PR[91,1] = PR[90,1] + 3.452;
   1:  PR[91,2] = PR[90,2] + 19.079;
   1:  PR[91,3] = PR[90,3] + 39.190;
   1:L PR[91] R[100]mm/sec CNT100;
   1:  PR[91,1] = PR[90,1] + 2.469;
   1:  PR[91,2] = PR[90,2] + 18.776;
   1:  PR[91,3] = PR[90,3] + 39.198;
   1:L PR[91] R[100]mm/sec CNT100;
   1:  PR[91,1] = PR[90,1] + 0.648;
   1:  PR[91,2] = PR[90,2] + 18.096;
   1:  PR[91,3] = PR[90,3] + 39.207;
   1:L PR[91] R[100]mm/sec CNT100;
   1:  PR[91,1] = PR[90,1] + 0.159;
   1:  PR[91,2] = PR[90,2] + 18.009;
   1:  PR[91,3] = PR[90,3] + 39.222;
   1:L PR[91] R[100]mm/sec CNT100;
   1:  PR[91,1] = PR[90,1] + -0.332;
   1:  PR[91,2] = PR[90,2] + 18.004;
   1:  PR[91,3] = PR[90,3] + 39.226;
   1:L PR[91] R[100]mm/sec CNT100;
   1:  PR[91,1] = PR[90,1] + -0.816;
   1:  PR[91,2] = PR[90,2] + 18.079;
   1:  PR[91,3] = PR[90,3] + 39.230;
   1:L PR[91] R[100]mm/sec CNT100;
   1:  PR[91,1] = PR[90,1] + -1.102;
   1:  PR[91,2] = PR[90,2] + 18.172;
   1:  PR[91,3] = PR[90,3] + 39.234;
   1:L PR[91] R[100]mm/sec CNT100;
   1:  PR[91,1] = PR[90,1] + -1.697;
   1:  PR[91,2] = PR[90,2] + 18.408;
   1:  PR[91,3] = PR[90,3] + 39.237;
   1:L PR[91] R[100]mm/sec CNT100;
   1:  PR[91,1] = PR[90,1] + -2.706;
   1:  PR[91,2] = PR[90,2] + 18.777;
   1:  PR[91,3] = PR[90,3] + 39.242;
   1:L PR[91] R[100]mm/sec CNT100;
   1:  PR[91,1] = PR[90,1] + -3.691;
   1:  PR[91,2] = PR[90,2] + 19.081;
   1:  PR[91,3] = PR[90,3] + 39.251;
   1:L PR[91] R[100]mm/sec CNT100;
